VAR_GLOBAL CONSTANT  (* DbmDescriptions *)
  gc_DbmTranslation_de_Text0 : WSTRING(39) := "Pressure Block Oscillation Sensor State";
  gc_DbmTranslation_de_Text1 : WSTRING(39) := "Pressure Block Oscillation Sensor Value";
  gc_DbmTranslation_de_Text2 : WSTRING(43) := "Pressure Block Oscillation Sensor Raw value";
  gc_DbmTranslation_de_Text3 : WSTRING(27) := "Pressure Brake Sensor State";
  gc_DbmTranslation_de_Text4 : WSTRING(27) := "Pressure Brake Sensor Value";
  gc_DbmTranslation_de_Text5 : WSTRING(31) := "Pressure Brake Sensor Raw value";
  gc_DbmTranslation_de_Text6 : WSTRING(37) := "Temperature Transmission Sensor State";
  gc_DbmTranslation_de_Text7 : WSTRING(37) := "Temperature Transmission Sensor Value";
  gc_DbmTranslation_de_Text8 : WSTRING(41) := "Temperature Transmission Sensor Raw value";
  gc_DbmTranslation_de_Text9 : WSTRING(25) := "Fault Pvg Left Trak State";
  gc_DbmTranslation_de_Text10 : WSTRING(29) := "Fault Pvg Left Trak Raw Value";
  gc_DbmTranslation_de_Text11 : WSTRING(26) := "Fault Pvg Right Trak State";
  gc_DbmTranslation_de_Text12 : WSTRING(30) := "Fault Pvg Right Trak Raw value";
  gc_DbmTranslation_de_Text13 : WSTRING(25) := "Down Axle oscillant State";
  gc_DbmTranslation_de_Text14 : WSTRING(39) := "Down Axle oscillant  Raw value pin 0 Nc";
  gc_DbmTranslation_de_Text15 : WSTRING(39) := "Down Axle oscillant  Raw value pin 1 No";
  gc_DbmTranslation_de_Text16 : WSTRING(20) := "Down Axle fixe state";
  gc_DbmTranslation_de_Text17 : WSTRING(24) := "Down Axle fixe Raw value";
  gc_DbmTranslation_de_Text18 : WSTRING(33) := "Down Axle fixe Raw value pin 1 No";
  gc_DbmTranslation_de_Text19 : WSTRING(23) := "Up Axle oscillant state";
  gc_DbmTranslation_de_Text20 : WSTRING(23) := "Up Axle oscillant value";
  gc_DbmTranslation_de_Text21 : WSTRING(18) := "Up Axle fixe state";
  gc_DbmTranslation_de_Text22 : WSTRING(22) := "Up Axle fixe raw value";
  gc_DbmTranslation_de_Text23 : WSTRING(29) := "Frame rotation sensor 1 state";
  gc_DbmTranslation_de_Text24 : WSTRING(33) := "Frame rotation sensor 1 raw value";
  gc_DbmTranslation_de_Text25 : WSTRING(39) := "Frame rotation sensor 1 raw value Pin 1";
  gc_DbmTranslation_de_Text26 : WSTRING(22) := "Rail hook sensor state";
  gc_DbmTranslation_de_Text27 : WSTRING(26) := "Rail hook sensor raw value";
  gc_DbmTranslation_de_Text28 : WSTRING(27) := "Inductive Rail sensor state";
  gc_DbmTranslation_de_Text29 : WSTRING(31) := "Inductive Rail sensor raw value";
  gc_DbmTranslation_de_Text30 : WSTRING(21) := "Centered turret state";
  gc_DbmTranslation_de_Text31 : WSTRING(25) := "Centered turret raw value";
  gc_DbmTranslation_de_Text32 : WSTRING(25) := "Work Key track Side state";
  gc_DbmTranslation_de_Text33 : WSTRING(29) := "Work Key track Side raw value";
  gc_DbmTranslation_de_Text34 : WSTRING(29) := "Frame rotation sensor 2 state";
  gc_DbmTranslation_de_Text35 : WSTRING(39) := "Frame rotation sensor 2 raw value Pin 0";
  gc_DbmTranslation_de_Text36 : WSTRING(39) := "Frame rotation sensor 2 raw value Pin 1";
  gc_DbmTranslation_de_Text37 : WSTRING(24) := "Work Key Bilateral state";
  gc_DbmTranslation_de_Text38 : WSTRING(28) := "Work Key Bilateral raw value";
  gc_DbmTranslation_de_Text39 : WSTRING(22) := "Work Key Centred state";
  gc_DbmTranslation_de_Text40 : WSTRING(26) := "Work Key Centred raw value";
  gc_DbmTranslation_de_Text41 : WSTRING(32) := "Abutment turret track side state";
  gc_DbmTranslation_de_Text42 : WSTRING(36) := "Abutment turret track side raw value";
  gc_DbmTranslation_de_Text43 : WSTRING(34) := "Abutment Turret Centred Side state";
  gc_DbmTranslation_de_Text44 : WSTRING(38) := "Abutment Turret Centred Side raw value";
  gc_DbmTranslation_de_Text45 : WSTRING(43) := "Oscillant Axle Speed Sensor Direction state";
  gc_DbmTranslation_de_Text46 : WSTRING(47) := "Oscillant Axle Speed Sensor Direction Raw value";
  gc_DbmTranslation_de_Text47 : WSTRING(38) := "Fixe Axle Speed Sensor Direction state";
  gc_DbmTranslation_de_Text48 : WSTRING(42) := "Fixe Axle Speed Sensor Direction Raw value";
  gc_DbmTranslation_de_Text49 : WSTRING(19) := "Trailer gache state";
  gc_DbmTranslation_de_Text50 : WSTRING(23) := "Trailer gache raw value";
  gc_DbmTranslation_de_Text51 : WSTRING(34) := "Measuring mast sensor folded state";
  gc_DbmTranslation_de_Text52 : WSTRING(38) := "Measuring mast sensor folded raw value";
  gc_DbmTranslation_de_Text53 : WSTRING(24) := "Oscillant Axle frequency";
  gc_DbmTranslation_de_Text54 : WSTRING(19) := "Fixe Axle frequency";
  gc_DbmTranslation_de_Text55 : WSTRING(25) := "Aru Radio 1 Contact state";
  gc_DbmTranslation_de_Text56 : WSTRING(29) := "Aru Radio 1 Contact raw value";
  gc_DbmTranslation_de_Text57 : WSTRING(25) := "Aru Radio 2 Contact state";
  gc_DbmTranslation_de_Text58 : WSTRING(29) := "Aru Radio 2 Contact raw value";
  gc_DbmTranslation_de_Text59 : WSTRING(19) := "Aru 1 Contact state";
  gc_DbmTranslation_de_Text60 : WSTRING(23) := "Aru 1 Contact raw value";
  gc_DbmTranslation_de_Text61 : WSTRING(19) := "Aru 2 Contact state";
  gc_DbmTranslation_de_Text62 : WSTRING(23) := "Aru 2 contact raw value";
  gc_DbmTranslation_de_Text63 : WSTRING(19) := "Starter motor state";
  gc_DbmTranslation_de_Text64 : WSTRING(23) := "Starter motor raw value";
  gc_DbmTranslation_de_Text65 : WSTRING(33) := "Autorisation High Speed Key State";
  gc_DbmTranslation_de_Text66 : WSTRING(37) := "Autorisation High Speed Key Raw Value";
  gc_DbmTranslation_de_Text67 : WSTRING(35) := "Electric pump Pressure Sensor State";
  gc_DbmTranslation_de_Text68 : WSTRING(35) := "Electric pump Pressure Sensor Value";
  gc_DbmTranslation_de_Text69 : WSTRING(39) := "Electric pump Pressure Sensor Raw value";
  gc_DbmTranslation_de_Text70 : WSTRING(29) := "Mast sensor position UP State";
  gc_DbmTranslation_de_Text71 : WSTRING(33) := "Mast sensor position UP Raw Value";
  gc_DbmTranslation_de_Text72 : WSTRING(46) := "Hydraulic valve uin down position sensor state";
  gc_DbmTranslation_de_Text73 : WSTRING(50) := "Hydraulic valve uin down position sensor raw value";
  gc_DbmTranslation_de_Text74 : WSTRING(33) := "Ev Deflector Transmission command";
  gc_DbmTranslation_de_Text75 : WSTRING(38) := "Ev Deflector Transmission actual value";
  gc_DbmTranslation_de_Text76 : WSTRING(28) := "Ev Up Measuring Mast command";
  gc_DbmTranslation_de_Text77 : WSTRING(33) := "Ev Up Measuring Mast actual value";
  gc_DbmTranslation_de_Text78 : WSTRING(30) := "Ev Down Measuring Mast command";
  gc_DbmTranslation_de_Text79 : WSTRING(35) := "Ev Down Measuring Mast actual value";
  gc_DbmTranslation_de_Text80 : WSTRING(30) := "Ev Service Brake Track command";
  gc_DbmTranslation_de_Text81 : WSTRING(35) := "Ev Service Brake Track actual value";
  gc_DbmTranslation_de_Text82 : WSTRING(26) := "Ev Power Reduction command";
  gc_DbmTranslation_de_Text83 : WSTRING(31) := "Ev Power Reduction actual value";
  gc_DbmTranslation_de_Text84 : WSTRING(27) := "Ev Frame Rotation 1 command";
  gc_DbmTranslation_de_Text85 : WSTRING(32) := "Ev Frame Rotation 1 actual value";
  gc_DbmTranslation_de_Text86 : WSTRING(27) := "Ev Frame Rotation 2 command";
  gc_DbmTranslation_de_Text87 : WSTRING(32) := "Ev Frame Rotation 2 actual value";
  gc_DbmTranslation_de_Text88 : WSTRING(29) := "Supply Radio Receiver command";
  gc_DbmTranslation_de_Text89 : WSTRING(34) := "Supply Radio Receiver actual value";
  gc_DbmTranslation_de_Text90 : WSTRING(34) := "Buzzer Lynx Moving Machine command";
  gc_DbmTranslation_de_Text91 : WSTRING(39) := "Buzzer Lynx Moving Machine actual value";
  gc_DbmTranslation_de_Text92 : WSTRING(28) := "White Lights Trailer command";
  gc_DbmTranslation_de_Text93 : WSTRING(33) := "White Lights Trailer actual value";
  gc_DbmTranslation_de_Text94 : WSTRING(26) := "Red Lights Trailer command";
  gc_DbmTranslation_de_Text95 : WSTRING(31) := "Red Lights Trailer actual value";
  gc_DbmTranslation_de_Text96 : WSTRING(23) := "White Light AVG command";
  gc_DbmTranslation_de_Text97 : WSTRING(28) := "White Light AVG actual value";
  gc_DbmTranslation_de_Text98 : WSTRING(23) := "White Light AVD command";
  gc_DbmTranslation_de_Text99 : WSTRING(28) := "White Light AVD actual value";
  gc_DbmTranslation_de_Text100 : WSTRING(21) := "Red Light AVG command";
  gc_DbmTranslation_de_Text101 : WSTRING(26) := "Red Light AVG actual value";
  gc_DbmTranslation_de_Text102 : WSTRING(21) := "Red Light AVD command";
  gc_DbmTranslation_de_Text103 : WSTRING(26) := "Red Light AVD actual value";
  gc_DbmTranslation_de_Text104 : WSTRING(23) := "White Light ARG command";
  gc_DbmTranslation_de_Text105 : WSTRING(28) := "White Light ARG actual value";
  gc_DbmTranslation_de_Text106 : WSTRING(23) := "White Light ARD command";
  gc_DbmTranslation_de_Text107 : WSTRING(28) := "White Light ARD actual value";
  gc_DbmTranslation_de_Text108 : WSTRING(21) := "Red Light ARG command";
  gc_DbmTranslation_de_Text109 : WSTRING(26) := "Red Light ARG actual value";
  gc_DbmTranslation_de_Text110 : WSTRING(21) := "Red Light ARD command";
  gc_DbmTranslation_de_Text111 : WSTRING(26) := "Red Light ARD actual value";
  gc_DbmTranslation_de_Text112 : WSTRING(29) := "Suplly Pvg Left Track command";
  gc_DbmTranslation_de_Text113 : WSTRING(34) := "Suplly Pvg Left Track actual value";
  gc_DbmTranslation_de_Text114 : WSTRING(30) := "Suplly Pvg Right Track command";
  gc_DbmTranslation_de_Text115 : WSTRING(35) := "Suplly Pvg Right Track actual value";
  gc_DbmTranslation_de_Text116 : WSTRING(33) := "Ev UnBlock Oscillation Axle state";
  gc_DbmTranslation_de_Text117 : WSTRING(40) := "Ev UnBlock Oscillation Axle command bool";
  gc_DbmTranslation_de_Text118 : WSTRING(26) := "Ev Up Axle Oscillant state";
  gc_DbmTranslation_de_Text119 : WSTRING(33) := "Ev Up Axle Oscillant Command Bool";
  gc_DbmTranslation_de_Text120 : WSTRING(29) := "Ev Down Axle Oscillant  state";
  gc_DbmTranslation_de_Text121 : WSTRING(35) := "Ev Down Axle Oscillant Command Bool";
  gc_DbmTranslation_de_Text122 : WSTRING(20) := "Ev Up AxleFixe state";
  gc_DbmTranslation_de_Text123 : WSTRING(28) := "Ev Up Axle Fixe Command Bool";
  gc_DbmTranslation_de_Text124 : WSTRING(22) := "Ev Down AxleFixe state";
  gc_DbmTranslation_de_Text125 : WSTRING(30) := "Ev Down Axle Fixe Command Bool";
  gc_DbmTranslation_de_Text126 : WSTRING(35) := "Ev Park Brake Axle Oscillant  state";
  gc_DbmTranslation_de_Text127 : WSTRING(42) := "Ev Park Brake Axle Oscillant  command bool";
  gc_DbmTranslation_de_Text128 : WSTRING(29) := "Ev Park Brake Axle Fixe state";
  gc_DbmTranslation_de_Text129 : WSTRING(37) := "Ev Park Brake Axle Fixe  command bool";
  gc_DbmTranslation_de_Text130 : WSTRING(37) := "Ev Service Brake Axle Oscillant state";
  gc_DbmTranslation_de_Text131 : WSTRING(36) := "Ev Service Brake Axle 1 command Bool";
  gc_DbmTranslation_de_Text132 : WSTRING(32) := "Ev Service Brake Axle Fixe state";
  gc_DbmTranslation_de_Text133 : WSTRING(36) := "Ev Service Brake Axle 2 command Bool";
  gc_DbmTranslation_de_Text134 : WSTRING(19) := "Klaxon Neotec state";
  gc_DbmTranslation_de_Text135 : WSTRING(26) := "Klaxon Neotec command bool";
  gc_DbmTranslation_de_Text136 : WSTRING(18) := "Forward pump state";
  gc_DbmTranslation_de_Text137 : WSTRING(21) := "Forward pump  command";
  gc_DbmTranslation_de_Text138 : WSTRING(27) := "Forward pump actual current";
  gc_DbmTranslation_de_Text139 : WSTRING(19) := "Backward pump state";
  gc_DbmTranslation_de_Text140 : WSTRING(22) := "Backward pump  command";
  gc_DbmTranslation_de_Text141 : WSTRING(28) := "Backward pump actual current";
  gc_DbmTranslation_de_Text142 : WSTRING(22) := "Pvg left track command";
  gc_DbmTranslation_de_Text143 : WSTRING(29) := "Pvg left track actual voltage";
  gc_DbmTranslation_de_Text144 : WSTRING(23) := "Pvg right track command";
  gc_DbmTranslation_de_Text145 : WSTRING(30) := "Pvg right track actual voltage";
  gc_DbmTranslation_de_Text146 : WSTRING(26) := "Supply Ana Sensors Command";
  gc_DbmTranslation_de_Text147 : WSTRING(24) := "Supply Ana Sensors Value";
  gc_DbmTranslation_de_Text148 : WSTRING(30) := "Pvg Left Track Lowside Command";
  gc_DbmTranslation_de_Text149 : WSTRING(28) := "Pvg Left Track Lowside Value";
  gc_DbmTranslation_de_Text150 : WSTRING(31) := "Pvg Right Track Lowside Command";
  gc_DbmTranslation_de_Text151 : WSTRING(29) := "Pvg Right Track Lowside Value";
  gc_DbmTranslation_de_Text152 : WSTRING(39) := "Return low side Ev Forward Pump command";
  gc_DbmTranslation_de_Text153 : WSTRING(37) := "Return low side Ev Forward Pump state";
  gc_DbmTranslation_de_Text154 : WSTRING(40) := "Return low side Ev Backward Pump command";
  gc_DbmTranslation_de_Text155 : WSTRING(38) := "Return low side Ev Backward Pump state";
  gc_DbmTranslation_de_Text156 : WSTRING(19) := "Neon Lights command";
  gc_DbmTranslation_de_Text157 : WSTRING(17) := "Neon Lights value";
  gc_DbmTranslation_de_Text158 : WSTRING(33) := "Ev 2 Deflector Transmission value";
  gc_DbmTranslation_de_Text159 : WSTRING(21) := "Cooling relay command";
  gc_DbmTranslation_de_Text160 : WSTRING(19) := "Cooling relay state";
  gc_DbmTranslation_de_Text161 : WSTRING(54) := "Sorties d’activation de l’Ev du deuxième frein de parc";
  gc_DbmTranslation_de_Text162 : WSTRING(54) := "Sorties d’activation de l’Ev du deuxième frein de parc";
  gc_DbmTranslation_de_Text163 : WSTRING(33) := "Ev 2nd Park Brake Axle Fixe State";
  gc_DbmTranslation_de_Text164 : WSTRING(33) := "Ev 2nd Park Brake Axle Osci State";
  gc_DbmTranslation_de_Text165 : WSTRING(41) := "Pvg Translation for Rail Electric Command";
  gc_DbmTranslation_de_Text166 : WSTRING(41) := "Pvg Translation for Rail Electric Voltage";
  gc_DbmTranslation_de_Text167 : WSTRING(48) := "Suplly Pvg Translation for Rail Electric Command";
  gc_DbmTranslation_de_Text168 : WSTRING(46) := "Suplly Pvg Translation for Rail Electric State";
  gc_DbmTranslation_de_Text169 : WSTRING(42) := "Ev Deviator for Rail Electric Mode Command";
  gc_DbmTranslation_de_Text170 : WSTRING(40) := "Ev Deviator for Rail Electric Mode State";
  gc_DbmTranslation_de_Text171 : WSTRING(43) := "Relay Cut Off Variator for Electric Command";
  gc_DbmTranslation_de_Text172 : WSTRING(41) := "Relay Cut Off Variator for Electric State";
  gc_DbmTranslation_de_Text173 : WSTRING(28) := "Relay Enable Battery Command";
  gc_DbmTranslation_de_Text174 : WSTRING(26) := "Relay Enable Battery State";
  gc_DbmTranslation_de_Text175 : WSTRING(25) := "Byte increased each cycle";
  gc_DbmTranslation_de_Text176 : WSTRING(22) := "Watchdog current state";
  gc_DbmTranslation_de_Text177 : WSTRING(11) := "Ecu voltage";
  gc_DbmTranslation_de_Text178 : WSTRING(13) := "Off Rail Mode";
  gc_DbmTranslation_de_Text179 : WSTRING(9) := "Rail Mode";
  gc_DbmTranslation_de_Text180 : WSTRING(75) := "Output value Lut of Manipulator left radio control in range -10000 to 10000";
  gc_DbmTranslation_de_Text181 : WSTRING(35) := "Output value Lut of Left Track Pvg ";
  gc_DbmTranslation_de_Text182 : WSTRING(76) := "Output value Lut of Manipulator Right radio control in range -10000 to 10000";
  gc_DbmTranslation_de_Text183 : WSTRING(36) := "Output value Lut of Right Track Pvg ";
  gc_DbmTranslation_de_Text184 : WSTRING(52) := "Outût value Lut of Joystick advance Rail translation";
  gc_DbmTranslation_de_Text185 : WSTRING(40) := "Output Lut  of Forward Pump Transmission";
  gc_DbmTranslation_de_Text186 : WSTRING(41) := "Output Lut  of Backward Pump Transmission";
  gc_DbmTranslation_de_Text187 : WSTRING(71) := "Calculate consigne current of Forward Pump transmission on percent *100";
  gc_DbmTranslation_de_Text188 : WSTRING(24) := "LastJoystickAdvanceValue";
  gc_DbmTranslation_de_Text189 : WSTRING(37) := "Scaling Value of Joystick advancement";
  gc_DbmTranslation_de_Text190 : WSTRING(39) := "State of service brake rail translation";
  gc_DbmTranslation_de_Text191 : WSTRING(36) := "Enable Start timer for service brake";
  gc_DbmTranslation_de_Text192 : WSTRING(48) := "Speed motor command provide by track transaltion";
  gc_DbmTranslation_de_Text193 : WSTRING(28) := "Force silent mode motor test";
  gc_DbmTranslation_de_Text194 : WSTRING(19) := "Angular sensor test";
  gc_DbmTranslation_de_Text195 : WSTRING(17) := "Speed axle sensor";
  gc_DbmTranslation_de_Text196 : WSTRING(18) := "Average Time cycle";
  gc_DbmTranslation_de_Text197 : WSTRING(14) := "Max time cycle";
  gc_DbmTranslation_de_Text198 : WSTRING(40) := "First translation for release park brake";
  gc_DbmTranslation_de_Text199 : WSTRING(35) := "Autorize Up Axle Oscillant movement";
  gc_DbmTranslation_de_Text200 : WSTRING(37) := "Autorize Down Axle Oscillant movement";
  gc_DbmTranslation_de_Text201 : WSTRING(30) := "Autorize Up Axle fixe movement";
  gc_DbmTranslation_de_Text202 : WSTRING(32) := "Autorize Down Axle fixe movement";
  gc_DbmTranslation_de_Text203 : WSTRING(19) := "Engine On run phase";
  gc_DbmTranslation_de_Text204 : WSTRING(74) := "Transaltion rail or off rail is solicited , flag send to C1 to pilot motor";
  gc_DbmTranslation_de_Text205 : WSTRING(42) := "Direction of rail translation (Av Ar Stop)";
  gc_DbmTranslation_de_Text206 : WSTRING(39) := "Set condition to active Aru radio alarm";
  gc_DbmTranslation_de_Text207 : WSTRING(36) := "Joystick advance setpoint after ramp";
  gc_DbmTranslation_de_Text208 : WSTRING(46) := "Stabilized stop flag to active park brake rail";
  gc_DbmTranslation_de_Text209 : WSTRING(48) := "Emergency brake flag to active sequence of brake";
  gc_DbmTranslation_de_Text210 : WSTRING(51) := "Flag when the timer emergency service brake is done";
  gc_DbmTranslation_de_Text211 : WSTRING(66) := "Flag when the timer stopped machine unblock osciilant axle is done";
  gc_DbmTranslation_de_Text212 : WSTRING(86) := "Output value Lut of Manipulator left radio control in range -10000 to 10000 after ramp";
  gc_DbmTranslation_de_Text213 : WSTRING(87) := "Output value Lut of Manipulator right radio control in range -10000 to 10000 after ramp";
  gc_DbmTranslation_de_Text214 : WSTRING(52) := "Delta beetwen left and right Pvg crawler advancement";
  gc_DbmTranslation_de_Text215 : WSTRING(65) := "Consigne left pvg track calcul with delta beetween left and right";
  gc_DbmTranslation_de_Text216 : WSTRING(66) := "Consigne right pvg track calcul with delta beetween left and right";
  gc_DbmTranslation_de_Text217 : WSTRING(56) := "Flag to detect brake when gachette or pedal are released";
  gc_DbmTranslation_de_Text218 : WSTRING(50) := "Counter for debug when alarm aru radio is detected";
  gc_DbmTranslation_de_Text219 : WSTRING(28) := "Red light ARG basket command";
  gc_DbmTranslation_de_Text220 : WSTRING(30) := "White light ARG basket command";
  gc_DbmTranslation_de_Text221 : WSTRING(32) := "Portilon close and ladder folded";
  gc_DbmTranslation_de_Text222 : WSTRING(46) := "Test boolean  command to refresh objet evision";
  gc_DbmTranslation_de_Text223 : WSTRING(60) := "Position of joysstick advancment ( AV_JOY, NEU_JOY , AR_JOY)";
  gc_DbmTranslation_de_Text224 : WSTRING(81) := "Retain position of joystick advancement , reset when brake sequence is sollicited";
  gc_DbmTranslation_de_Text225 : WSTRING(37) := "Authorize forward crawler translation";
  gc_DbmTranslation_de_Text226 : WSTRING(38) := "Authorize backward crawler translation";
  gc_DbmTranslation_de_Text227 : WSTRING(22) := "Return value uart init";
  gc_DbmTranslation_de_Text228 : WSTRING(35) := "Authorize translation rail movement";
  gc_DbmTranslation_de_Text229 : WSTRING(25) := "Ev forward track consigne";
  gc_DbmTranslation_de_Text230 : WSTRING(24) := "Ev forward rail consigne";
  gc_DbmTranslation_de_Text231 : WSTRING(0) := "";
  gc_DbmTranslation_de_Text232 : WSTRING(21) := "Variable debug Neotec";
  gc_DbmTranslation_de_Text233 : WSTRING(21) := "Variable debug Neotec";
  gc_DbmTranslation_de_Text234 : WSTRING(21) := "Variable debug Neotec";
  gc_DbmTranslation_de_Text235 : WSTRING(21) := "Variable debug Neotec";
  gc_DbmTranslation_de_Text236 : WSTRING(21) := "Variable debug Neotec";
  gc_DbmTranslation_de_Text237 : WSTRING(21) := "Variable debug Neotec";
  gc_DbmTranslation_de_Text238 : WSTRING(21) := "Variable debug Neotec";
  gc_DbmTranslation_de_Text239 : WSTRING(21) := "Variable debug Neotec";
  gc_DbmTranslation_de_Text240 : WSTRING(21) := "Variable debug Neotec";
  gc_DbmTranslation_de_Text241 : WSTRING(21) := "Variable debug Neotec";
  gc_DbmTranslation_de_Text242 : WSTRING(21) := "Variable debug Neotec";
  gc_DbmTranslation_de_Text243 : WSTRING(21) := "Variable debug Neotec";
  gc_DbmTranslation_de_Text244 : WSTRING(21) := "Variable debug Neotec";
  gc_DbmTranslation_de_Text245 : WSTRING(21) := "Variable debug Neotec";
  gc_DbmTranslation_de_Text246 : WSTRING(21) := "Variable debug Neotec";
  gc_DbmTranslation_de_Text247 : WSTRING(21) := "Variable debug Neotec";
  gc_DbmTranslation_de_Text248 : WSTRING(21) := "Variable debug Neotec";
  gc_DbmTranslation_de_Text249 : WSTRING(21) := "Variable debug Neotec";
  gc_DbmTranslation_de_Text250 : WSTRING(21) := "Variable debug Neotec";
  gc_DbmTranslation_de_Text251 : WSTRING(21) := "Variable debug Neotec";
  gc_DbmTranslation_de_Text252 : WSTRING(21) := "Variable debug Neotec";
  gc_DbmTranslation_de_Text253 : WSTRING(21) := "Variable debug Neotec";
  gc_DbmTranslation_de_Text254 : WSTRING(21) := "Variable debug Neotec";
  gc_DbmTranslation_de_Text255 : WSTRING(21) := "Variable debug Neotec";
  gc_DbmTranslation_de_Text256 : WSTRING(21) := "Variable debug Neotec";
  gc_DbmTranslation_de_Text257 : WSTRING(21) := "Variable debug Neotec";
  gc_DbmTranslation_de_Text258 : WSTRING(21) := "Variable debug Neotec";
  gc_DbmTranslation_de_Text259 : WSTRING(21) := "Variable debug Neotec";
  gc_DbmTranslation_de_Text260 : WSTRING(21) := "Variable debug Neotec";
  gc_DbmTranslation_de_Text261 : WSTRING(21) := "Variable debug Neotec";
  gc_DbmTranslation_de_Text262 : WSTRING(21) := "Variable debug Neotec";
  gc_DbmTranslation_de_Text263 : WSTRING(21) := "Variable debug Neotec";
  gc_DbmTranslation_de_Text264 : WSTRING(21) := "Variable debug Neotec";
  gc_DbmTranslation_de_Text265 : WSTRING(21) := "Variable debug Neotec";
  gc_DbmTranslation_de_Text266 : WSTRING(21) := "Variable debug Neotec";
  gc_DbmTranslation_de_Text267 : WSTRING(21) := "Variable debug Neotec";
  gc_DbmTranslation_de_Text268 : WSTRING(21) := "Variable debug Neotec";
  gc_DbmTranslation_de_Text269 : WSTRING(21) := "Variable debug Neotec";
  gc_DbmTranslation_de_Text270 : WSTRING(21) := "Variable debug Neotec";
  gc_DbmTranslation_de_Text271 : WSTRING(21) := "Variable debug Neotec";
  gc_DbmTranslation_de_Text272 : WSTRING(28) := "Red light ARD basket command";
  gc_DbmTranslation_de_Text273 : WSTRING(30) := "White light ARD basket command";
  gc_DbmTranslation_de_Text274 : WSTRING(26) := "Active failure is detected";
  gc_DbmTranslation_de_Text275 : WSTRING(19) := "Reduction pump rail";
  gc_DbmTranslation_de_Text276 : WSTRING(20) := "Reduction pump track";
  gc_DbmTranslation_de_Text277 : WSTRING(25) := "Active white lights 15746";
  gc_DbmTranslation_de_Text278 : WSTRING(24) := "White light Av 15746 Cmd";
  gc_DbmTranslation_de_Text279 : WSTRING(24) := "White light Ar 15746 Cmd";
  gc_DbmTranslation_de_Text280 : WSTRING(38) := "Shunt all logic to test electricall IO";
  gc_DbmTranslation_de_Text281 : WSTRING(29) := "Send Event Datalogger Message";
  gc_DbmTranslation_de_Text282 : WSTRING(21) := "Depend de l’option MG";
  gc_DbmTranslation_de_Text283 : WSTRING(13) := "Slow Blinking";
  gc_DbmTranslation_de_Text284 : WSTRING(14) := "Total distance";
  gc_DbmTranslation_de_Text285 : WSTRING(19) := "Running Stable 48XS";
  gc_DbmTranslation_de_Text286 : WSTRING(39) := "Alarm Hydraulic Temperature Rail Active";
  gc_DbmTranslation_de_Text287 : WSTRING(42) := "Alarm Hydraulic Temperature Crawler Active";
  gc_DbmTranslation_de_Text288 : WSTRING(17) := "Diag Faulty Value";
  gc_DbmTranslation_de_Text289 : WSTRING(15) := "Diag Device Num";
  gc_DbmTranslation_de_Text290 : WSTRING(15) := "Diag Error Code";
  gc_DbmTranslation_de_Text291 : WSTRING(21) := "Engine running stable";
  gc_DbmTranslation_de_Text292 : WSTRING(42) := "Select config hollandaise to control light";
  gc_DbmTranslation_de_Text293 : WSTRING(37) := "Portillon is installed on the machine";
  gc_DbmTranslation_de_Text294 : WSTRING(34) := "Ladder is installed on the machine";
  gc_DbmTranslation_de_Text295 : WSTRING(41) := "Measuring mat is installed on the machine";
  gc_DbmTranslation_de_Text296 : WSTRING(107) := "-SpeedMaxRail Acces Site- Inclinaison Baslet most be in low sector for acces site speed on translation rail";
  gc_DbmTranslation_de_Text297 : WSTRING(90) := "-SpeedMaxRail Acces Site- Basket most be centered for acces site speed on translation rail";
  gc_DbmTranslation_de_Text298 : WSTRING(64) := "The digital display o the measuring mast is used on this vehicle";
  gc_DbmTranslation_de_Text299 : WSTRING(30) := "Autorisation work key present ";
  gc_DbmTranslation_de_Text300 : WSTRING(40) := "Option d’activation du mode double frein";
  gc_DbmTranslation_de_Text301 : WSTRING(50) := "Strukton configuration for new performance machine";
  gc_DbmTranslation_de_Text302 : WSTRING(46) := "Basket and turret limited by a mechanical stop";
  gc_DbmTranslation_de_Text303 : WSTRING(24) := "Presence of sensor plate";
  gc_DbmTranslation_de_Text304 : WSTRING(29) := "Number of brake cycle perform";
  gc_DbmTranslation_de_Text305 : WSTRING(10) := "Light mode";
  gc_DbmTranslation_de_Text306 : WSTRING(0) := "";
  gc_DbmTranslation_de_Text307 : WSTRING(0) := "";
  gc_DbmTranslation_de_Text308 : WSTRING(0) := "";
  gc_DbmTranslation_de_Text309 : WSTRING(0) := "";
  gc_DbmTranslation_de_Text310 : WSTRING(0) := "";
  gc_DbmTranslation_de_Text311 : WSTRING(0) := "";
  gc_DbmTranslation_de_Text312 : WSTRING(0) := "";
  gc_DbmTranslation_de_Text313 : WSTRING(0) := "";
  gc_DbmTranslation_de_Text314 : WSTRING(0) := "";
  gc_DbmTranslation_de_Text315 : WSTRING(0) := "";
  gc_DbmTranslation_de_Text316 : WSTRING(0) := "";
  gc_DbmTranslation_de_Text317 : WSTRING(0) := "";
  gc_DbmTranslation_de_Text318 : WSTRING(0) := "";
  gc_DbmTranslation_de_Text319 : WSTRING(0) := "";
  gc_DbmTranslation_de_Text320 : WSTRING(0) := "";
  gc_DbmTranslation_de_Text321 : WSTRING(54) := "Nombres de cycle de frein pour les freins additionnels";
  gc_DbmTranslation_de_Text322 : WSTRING(18) := "Total Distance Msb";
  gc_DbmTranslation_de_Text323 : WSTRING(18) := "Total Distance Lsb";
  gc_DbmTranslation_de_Text324 : WSTRING(77) := "Limit threshold of angle to stop movement , angular sensor from radio control";
  gc_DbmTranslation_de_Text325 : WSTRING(43) := "Treshold minimal speed to active park brake";
  gc_DbmTranslation_de_Text326 : WSTRING(46) := "Treshold minimal speed to active service brake";
  gc_DbmTranslation_de_Text327 : WSTRING(41) := "Additionnal Pourcent Forward Pump Command";
  gc_DbmTranslation_de_Text328 : WSTRING(67) := "Additionnal Pourcent Forward Pump Command when sient mode is active";
  gc_DbmTranslation_de_Text329 : WSTRING(21) := "Node Id radio command";
  gc_DbmTranslation_de_Text330 : WSTRING(34) := "Dead Zone joystick rotation turret";
  gc_DbmTranslation_de_Text331 : WSTRING(52) := "Timer before 2nd Service Axle brake rail translation";
  gc_DbmTranslation_de_Text332 : WSTRING(26) := "Time Service Brake Offrail";
  gc_DbmTranslation_de_Text333 : WSTRING(59) := "Ev Forward Pump - PWM output parameters- engine off current";
  gc_DbmTranslation_de_Text334 : WSTRING(56) := "Ev Forward Pump - PWM output parameters- minimal current";
  gc_DbmTranslation_de_Text335 : WSTRING(54) := "Ev Forward Pump - PWM output parameters- stop current ";
  gc_DbmTranslation_de_Text336 : WSTRING(60) := "Ev Backward Pump - PWM output parameters- engine off current";
  gc_DbmTranslation_de_Text337 : WSTRING(57) := "Ev Backward Pump - PWM output parameters- minimal current";
  gc_DbmTranslation_de_Text338 : WSTRING(55) := "Ev Backward Pump - PWM output parameters- stop current ";
  gc_DbmTranslation_de_Text339 : WSTRING(67) := "Position neutral of joystick advancement regarding batterie voltage";
  gc_DbmTranslation_de_Text340 : WSTRING(46) := "PID - Ev Forward Pump - Gp - proportional gain";
  gc_DbmTranslation_de_Text341 : WSTRING(54) := "PID - Ev Forward Pump - Ti - integration time constant";
  gc_DbmTranslation_de_Text342 : WSTRING(53) := "PID - Ev Forward Pump - Td - derivation time constant";
  gc_DbmTranslation_de_Text343 : WSTRING(46) := "PID - Ev Forward Pump - Gp - proportional gain";
  gc_DbmTranslation_de_Text344 : WSTRING(54) := "PID - Ev Forward Pump - Ti - integration time constant";
  gc_DbmTranslation_de_Text345 : WSTRING(53) := "PID - Ev Forward Pump - Td - derivation time constant";
  gc_DbmTranslation_de_Text346 : WSTRING(80) := "PressureBlockOscillationSensor - input current - output characteristic - Positif";
  gc_DbmTranslation_de_Text347 : WSTRING(80) := "PressureBlockOscillationSensor - input current - output characteristic - Neutral";
  gc_DbmTranslation_de_Text348 : WSTRING(80) := "PressureBlockOscillationSensor - input current - output characteristic - Negatif";
  gc_DbmTranslation_de_Text349 : WSTRING(69) := "PressureBrakeSensor - input current - output characteristic - Positif";
  gc_DbmTranslation_de_Text350 : WSTRING(69) := "PressureBrakeSensor - input current - output characteristic - Neutral";
  gc_DbmTranslation_de_Text351 : WSTRING(69) := "PressureBrakeSensor - input current - output characteristic - Negatif";
  gc_DbmTranslation_de_Text352 : WSTRING(79) := "TemperatureTransmissionSensor - input current - output characteristic - Positif";
  gc_DbmTranslation_de_Text353 : WSTRING(79) := "TemperatureTransmissionSensor - input current - output characteristic - Neutral";
  gc_DbmTranslation_de_Text354 : WSTRING(79) := "TemperatureTransmissionSensor - input current - output characteristic - Negatif";
  gc_DbmTranslation_de_Text355 : WSTRING(55) := "Consigne min Ev forward apply with joystick advancement";
  gc_DbmTranslation_de_Text356 : WSTRING(55) := "Consigne max Ev forward apply with joystick advancement";
  gc_DbmTranslation_de_Text357 : WSTRING(56) := "Consigne min Ev backward apply with joystick advancement";
  gc_DbmTranslation_de_Text358 : WSTRING(56) := "Consigne max Ev backward apply with joystick advancement";
  gc_DbmTranslation_de_Text359 : WSTRING(96) := "Time  ramp to Ev rail [0] Pos incr time, [1] Pos decr time,[2] Neg incr time , [3] Neg decr time";
  gc_DbmTranslation_de_Text360 : WSTRING(96) := "Time  ramp to Ev rail [0] Pos incr time, [1] Pos decr time,[2] Neg incr time , [3] Neg decr time";
  gc_DbmTranslation_de_Text361 : WSTRING(96) := "Time  ramp to Ev rail [0] Pos incr time, [1] Pos decr time,[2] Neg incr time , [3] Neg decr time";
  gc_DbmTranslation_de_Text362 : WSTRING(96) := "Time  ramp to Ev rail [0] Pos incr time, [1] Pos decr time,[2] Neg incr time , [3] Neg decr time";
  gc_DbmTranslation_de_Text363 : WSTRING(96) := "Time  ramp to Ev rail [0] Pos incr time, [1] Pos decr time,[2] Neg incr time , [3] Neg decr time";
  gc_DbmTranslation_de_Text364 : WSTRING(53) := "Consigne min Ev forward apply for crawler advancement";
  gc_DbmTranslation_de_Text365 : WSTRING(53) := "Consigne max Ev forward apply for crawler advancement";
  gc_DbmTranslation_de_Text366 : WSTRING(72) := "Ratio apply to ramp signal to control Ev forward for crawler advancement";
  gc_DbmTranslation_de_Text367 : WSTRING(72) := "Ratio apply to ramp signal to control Ev forward for crawler advancement";
  gc_DbmTranslation_de_Text368 : WSTRING(72) := "Ratio apply to ramp signal to control Ev forward for crawler advancement";
  gc_DbmTranslation_de_Text369 : WSTRING(69) := "Park Brake rail - Treshold of regime motor to active park brake rail ";
  gc_DbmTranslation_de_Text370 : WSTRING(95) := "Consigne min Pvg Left Track apply when mapinulator get out neutral position to forward position";
  gc_DbmTranslation_de_Text371 : WSTRING(30) := "Consigne max Pvg Left Track Av";
  gc_DbmTranslation_de_Text372 : WSTRING(96) := "Consigne min Pvg Left Track apply when mapinulator get out neutral position to backward position";
  gc_DbmTranslation_de_Text373 : WSTRING(30) := "Consigne max Pvg Left Track Ar";
  gc_DbmTranslation_de_Text374 : WSTRING(96) := "Consigne min Pvg Right Track apply when mapinulator get out neutral position to forward position";
  gc_DbmTranslation_de_Text375 : WSTRING(31) := "Consigne max Pvg Right Track Av";
  gc_DbmTranslation_de_Text376 : WSTRING(97) := "Consigne min Pvg Right Track apply when mapinulator get out neutral position to backward position";
  gc_DbmTranslation_de_Text377 : WSTRING(31) := "Consigne max Pvg Right Track Ar";
  gc_DbmTranslation_de_Text378 : WSTRING(105) := "Time  ramp apply to left track [0] Pos incr time, [1] Pos decr time,[2] Neg incr time , [3] Neg decr time";
  gc_DbmTranslation_de_Text379 : WSTRING(105) := "Time  ramp apply to left track [0] Pos incr time, [1] Pos decr time,[2] Neg incr time , [3] Neg decr time";
  gc_DbmTranslation_de_Text380 : WSTRING(105) := "Time  ramp apply to left track [0] Pos incr time, [1] Pos decr time,[2] Neg incr time , [3] Neg decr time";
  gc_DbmTranslation_de_Text381 : WSTRING(105) := "Time  ramp apply to left track [0] Pos incr time, [1] Pos decr time,[2] Neg incr time , [3] Neg decr time";
  gc_DbmTranslation_de_Text382 : WSTRING(105) := "Time  ramp apply to left track [0] Pos incr time, [1] Pos decr time,[2] Neg incr time , [3] Neg decr time";
  gc_DbmTranslation_de_Text383 : WSTRING(106) := "Time  ramp apply to right track [0] Pos incr time, [1] Pos decr time,[2] Neg incr time , [3] Neg decr time";
  gc_DbmTranslation_de_Text384 : WSTRING(106) := "Time  ramp apply to right track [0] Pos incr time, [1] Pos decr time,[2] Neg incr time , [3] Neg decr time";
  gc_DbmTranslation_de_Text385 : WSTRING(106) := "Time  ramp apply to right track [0] Pos incr time, [1] Pos decr time,[2] Neg incr time , [3] Neg decr time";
  gc_DbmTranslation_de_Text386 : WSTRING(106) := "Time  ramp apply to right track [0] Pos incr time, [1] Pos decr time,[2] Neg incr time , [3] Neg decr time";
  gc_DbmTranslation_de_Text387 : WSTRING(106) := "Time  ramp apply to right track [0] Pos incr time, [1] Pos decr time,[2] Neg incr time , [3] Neg decr time";
  gc_DbmTranslation_de_Text388 : WSTRING(38) := "Time to detect stabilized stop machine";
  gc_DbmTranslation_de_Text389 : WSTRING(67) := "Treshold low spped to start timer to detect stabilized stop machine";
  gc_DbmTranslation_de_Text390 : WSTRING(66) := "Time before release service brake when emergency brake is detected";
  gc_DbmTranslation_de_Text391 : WSTRING(57) := "Time stopped machine to controle unblock oscillation axle";
  gc_DbmTranslation_de_Text392 : WSTRING(87) := "Low treshold speed of oscillation and fixe axle to start timer unblock oscillation axle";
  gc_DbmTranslation_de_Text393 : WSTRING(55) := "Gap max beetween left and right Pvg crawler advancement";
  gc_DbmTranslation_de_Text394 : WSTRING(84) := "Gap max beetween left and right Pvg crawler advancement when manipulator is inverted";
  gc_DbmTranslation_de_Text395 : WSTRING(36) := "Treshold Ana to bool input from 48xs";
  gc_DbmTranslation_de_Text396 : WSTRING(65) := "In min joystick advancement pourcentent by 10 of batterie voltage";
  gc_DbmTranslation_de_Text397 : WSTRING(65) := "In max joystick advancement pourcentent by 10 of batterie voltage";
  gc_DbmTranslation_de_Text398 : WSTRING(35) := "Speed mini treshol to re authorise ";
  gc_DbmTranslation_de_Text399 : WSTRING(44) := "Number element for average slope trans angle";
  gc_DbmTranslation_de_Text400 : WSTRING(43) := "Number element for average slope long angle";
  gc_DbmTranslation_de_Text401 : WSTRING(35) := "Dead zone joystick rail advancement";
  gc_DbmTranslation_de_Text402 : WSTRING(57) := "Number element for average slope trans angle 2nd channels";
  gc_DbmTranslation_de_Text403 : WSTRING(56) := "Number element for average slope long angle 2nd channels";
  gc_DbmTranslation_de_Text404 : WSTRING(18) := "Param debug Neotec";
  gc_DbmTranslation_de_Text405 : WSTRING(18) := "Param debug Neotec";
  gc_DbmTranslation_de_Text406 : WSTRING(18) := "Param debug Neotec";
  gc_DbmTranslation_de_Text407 : WSTRING(18) := "Param debug Neotec";
  gc_DbmTranslation_de_Text408 : WSTRING(18) := "Param debug Neotec";
  gc_DbmTranslation_de_Text409 : WSTRING(18) := "Param debug Neotec";
  gc_DbmTranslation_de_Text410 : WSTRING(18) := "Param debug Neotec";
  gc_DbmTranslation_de_Text411 : WSTRING(18) := "Param debug Neotec";
  gc_DbmTranslation_de_Text412 : WSTRING(18) := "Param debug Neotec";
  gc_DbmTranslation_de_Text413 : WSTRING(18) := "Param debug Neotec";
  gc_DbmTranslation_de_Text414 : WSTRING(18) := "Param debug Neotec";
  gc_DbmTranslation_de_Text415 : WSTRING(18) := "Param debug Neotec";
  gc_DbmTranslation_de_Text416 : WSTRING(18) := "Param debug Neotec";
  gc_DbmTranslation_de_Text417 : WSTRING(18) := "Param debug Neotec";
  gc_DbmTranslation_de_Text418 : WSTRING(18) := "Param debug Neotec";
  gc_DbmTranslation_de_Text419 : WSTRING(18) := "Param debug Neotec";
  gc_DbmTranslation_de_Text420 : WSTRING(18) := "Param debug Neotec";
  gc_DbmTranslation_de_Text421 : WSTRING(57) := "Treshold hydraulique temperature to control cooling relay";
  gc_DbmTranslation_de_Text422 : WSTRING(22) := "Time to control cooler";
  gc_DbmTranslation_de_Text423 : WSTRING(37) := "Time fault pressure reduction crawler";
  gc_DbmTranslation_de_Text424 : WSTRING(35) := "Rail joystick ratio two speed fault";
  gc_DbmTranslation_de_Text425 : WSTRING(25) := "Timeout sdo resquest time";
  gc_DbmTranslation_de_Text426 : WSTRING(29) := "Period Blinck off White Light";
  gc_DbmTranslation_de_Text427 : WSTRING(48) := "filtrage et le lissage de la valeur du joystick.";
  gc_DbmTranslation_de_Text428 : WSTRING(92) := "temporisation de l’AU afin d’attendre la fin des rampes avec un freinage d’urgence (Mode MG)";
  gc_DbmTranslation_de_Text429 : WSTRING(59) := "seuil d’angle tourelle pour la petite vitesse, côté positif";
  gc_DbmTranslation_de_Text430 : WSTRING(59) := "seuil d’angle tourelle pour la petite vitesse, côté négatif";
  gc_DbmTranslation_de_Text431 : WSTRING(25) := "Number of file parameters";
  gc_DbmTranslation_de_Text432 : WSTRING(13) := "Version Major";
  gc_DbmTranslation_de_Text433 : WSTRING(14) := "Version Minior";
  gc_DbmTranslation_de_Text434 : WSTRING(13) := "Version Patch";
  gc_DbmTranslation_de_Text435 : WSTRING(14) := "Version Custom";
  gc_DbmTranslation_de_Text436 : WSTRING(76) := "ElectricPumpPressureSensor - input current - output characteristic - Positif";
  gc_DbmTranslation_de_Text437 : WSTRING(76) := "ElectricPumpPressureSensor - input current - output characteristic - Neutral";
  gc_DbmTranslation_de_Text438 : WSTRING(76) := "ElectricPumpPressureSensor - input current - output characteristic - Negatif";
  gc_DbmTranslation_de_Text439 : WSTRING(44) := "Max point Lut Manipulator Left radio control";
  gc_DbmTranslation_de_Text440 : WSTRING(52) := "Lut array X value for Manipulator Left radio control";
  gc_DbmTranslation_de_Text441 : WSTRING(52) := "Lut array X value for Manipulator Left radio control";
  gc_DbmTranslation_de_Text442 : WSTRING(52) := "Lut array X value for Manipulator Left radio control";
  gc_DbmTranslation_de_Text443 : WSTRING(52) := "Lut array Y value for Manipulator Left radio control";
  gc_DbmTranslation_de_Text444 : WSTRING(52) := "Lut array Y value for Manipulator Left radio control";
  gc_DbmTranslation_de_Text445 : WSTRING(52) := "Lut array Y value for Manipulator Left radio control";
  gc_DbmTranslation_de_Text446 : WSTRING(45) := "Max point Lut Manipulator Right radio control";
  gc_DbmTranslation_de_Text447 : WSTRING(53) := "Lut array X value for Manipulator Right radio control";
  gc_DbmTranslation_de_Text448 : WSTRING(53) := "Lut array X value for Manipulator Right radio control";
  gc_DbmTranslation_de_Text449 : WSTRING(53) := "Lut array X value for Manipulator Right radio control";
  gc_DbmTranslation_de_Text450 : WSTRING(53) := "Lut array Y value for Manipulator Right radio control";
  gc_DbmTranslation_de_Text451 : WSTRING(53) := "Lut array Y value for Manipulator Right radio control";
  gc_DbmTranslation_de_Text452 : WSTRING(53) := "Lut array Y value for Manipulator Right radio control";
  gc_DbmTranslation_de_Text453 : WSTRING(40) := "Max point Lut for Left track pvg command";
  gc_DbmTranslation_de_Text454 : WSTRING(25) := "Left track Pvg Ramp ratio";
  gc_DbmTranslation_de_Text455 : WSTRING(25) := "Left track Pvg Ramp ratio";
  gc_DbmTranslation_de_Text456 : WSTRING(25) := "Left track Pvg Ramp ratio";
  gc_DbmTranslation_de_Text457 : WSTRING(50) := "Range value of left track Pvg apply to ramp signal";
  gc_DbmTranslation_de_Text458 : WSTRING(50) := "Range value of left track Pvg apply to ramp signal";
  gc_DbmTranslation_de_Text459 : WSTRING(50) := "Range value of left track Pvg apply to ramp signal";
  gc_DbmTranslation_de_Text460 : WSTRING(50) := "Range value of left track Pvg apply to ramp signal";
  gc_DbmTranslation_de_Text461 : WSTRING(26) := "Right track Pvg Ramp ratio";
  gc_DbmTranslation_de_Text462 : WSTRING(26) := "Right track Pvg Ramp ratio";
  gc_DbmTranslation_de_Text463 : WSTRING(26) := "Right track Pvg Ramp ratio";
  gc_DbmTranslation_de_Text464 : WSTRING(51) := "Range value of right track Pvg apply to ramp signal";
  gc_DbmTranslation_de_Text465 : WSTRING(51) := "Range value of right track Pvg apply to ramp signal";
  gc_DbmTranslation_de_Text466 : WSTRING(51) := "Range value of right track Pvg apply to ramp signal";
  gc_DbmTranslation_de_Text467 : WSTRING(51) := "Range value of right track Pvg apply to ramp signal";
  gc_DbmTranslation_de_Text468 : WSTRING(56) := "Max point Lut Forward pump transmission rail translation";
  gc_DbmTranslation_de_Text469 : WSTRING(64) := "Lut array X value for Forward pump transmission rail translation";
  gc_DbmTranslation_de_Text470 : WSTRING(64) := "Lut array X value for Forward pump transmission rail translation";
  gc_DbmTranslation_de_Text471 : WSTRING(64) := "Lut array X value for Forward pump transmission rail translation";
  gc_DbmTranslation_de_Text472 : WSTRING(64) := "Lut array Y value for Forward pump transmission rail translation";
  gc_DbmTranslation_de_Text473 : WSTRING(64) := "Lut array Y value for Forward pump transmission rail translation";
  gc_DbmTranslation_de_Text474 : WSTRING(64) := "Lut array Y value for Forward pump transmission rail translation";
  gc_DbmTranslation_de_Text475 : WSTRING(57) := "Max point Lut Backward pump transmission rail translation";
  gc_DbmTranslation_de_Text476 : WSTRING(64) := "Lut array X value for Backwardpump transmission rail translation";
  gc_DbmTranslation_de_Text477 : WSTRING(64) := "Lut array X value for Backwardpump transmission rail translation";
  gc_DbmTranslation_de_Text478 : WSTRING(64) := "Lut array X value for Backwardpump transmission rail translation";
  gc_DbmTranslation_de_Text479 : WSTRING(64) := "Lut array Y value for Backwardpump transmission rail translation";
  gc_DbmTranslation_de_Text480 : WSTRING(64) := "Lut array Y value for Backwardpump transmission rail translation";
  gc_DbmTranslation_de_Text481 : WSTRING(64) := "Lut array Y value for Backwardpump transmission rail translation";
  gc_DbmTranslation_de_Text482 : WSTRING(36) := "Forward pump transmission Ramp ratio";
  gc_DbmTranslation_de_Text483 : WSTRING(36) := "Forward pump transmission Ramp ratio";
  gc_DbmTranslation_de_Text484 : WSTRING(36) := "Forward pump transmission Ramp ratio";
  gc_DbmTranslation_de_Text485 : WSTRING(51) := "Range value of Forward pump transmission Ramp ratio";
  gc_DbmTranslation_de_Text486 : WSTRING(51) := "Range value of Forward pump transmission Ramp ratio";
  gc_DbmTranslation_de_Text487 : WSTRING(51) := "Range value of Forward pump transmission Ramp ratio";
  gc_DbmTranslation_de_Text488 : WSTRING(51) := "Range value of Forward pump transmission Ramp ratio";
  gc_DbmTranslation_de_Text489 : WSTRING(37) := "Backward pump transmission Ramp ratio";
  gc_DbmTranslation_de_Text490 : WSTRING(37) := "Backward pump transmission Ramp ratio";
  gc_DbmTranslation_de_Text491 : WSTRING(37) := "Backward pump transmission Ramp ratio";
  gc_DbmTranslation_de_Text492 : WSTRING(52) := "Range value of Backward pump transmission Ramp ratio";
  gc_DbmTranslation_de_Text493 : WSTRING(52) := "Range value of Backward pump transmission Ramp ratio";
  gc_DbmTranslation_de_Text494 : WSTRING(52) := "Range value of Backward pump transmission Ramp ratio";
  gc_DbmTranslation_de_Text495 : WSTRING(52) := "Range value of Backward pump transmission Ramp ratio";
  gc_DbmTranslation_de_Text496 : WSTRING(38) := "Offset apply to calcul angle of turret";
  gc_DbmTranslation_de_Text497 : WSTRING(55) := "Slope Long offset to calibrate value of longetude angle";
  gc_DbmTranslation_de_Text498 : WSTRING(58) := "Slope Trans offset to calibrate value of transversal angle";
  gc_DbmTranslation_de_Text499 : WSTRING(68) := "Slope Long offset to calibrate value of longetude angle 2nd channels";
  gc_DbmTranslation_de_Text500 : WSTRING(71) := "Slope Trans offset to calibrate value of transversal angle 2nd channels";
  gc_DbmTranslation_de_Text501 : WSTRING(53) := "Offset apply to calcul angle of turret second channel";
  gc_DbmTranslation_de_Text502 : WSTRING(21) := "Encodeur Turret Msb 1";
  gc_DbmTranslation_de_Text503 : WSTRING(21) := "Encodeur Turret Msb 2";
  gc_DbmTranslation_de_Text504 : WSTRING(21) := "Encodeur Turret Lsb 1";
  gc_DbmTranslation_de_Text505 : WSTRING(21) := "Encodeur Turret Lsb 2";
  gc_DbmTranslation_de_Text506 : WSTRING(29) := "Up  Inclinaison basket button";
  gc_DbmTranslation_de_Text507 : WSTRING(40) := "Up  Inclinaison basket  button raw value";
  gc_DbmTranslation_de_Text508 : WSTRING(31) := "Down  Inclinaison basket button";
  gc_DbmTranslation_de_Text509 : WSTRING(41) := "Down  Inclinaison basket button raw value";
  gc_DbmTranslation_de_Text510 : WSTRING(18) := "Up pendular button";
  gc_DbmTranslation_de_Text511 : WSTRING(28) := "Up pendular button raw value";
  gc_DbmTranslation_de_Text512 : WSTRING(20) := "Down pendular button";
  gc_DbmTranslation_de_Text513 : WSTRING(30) := "Down pendular button raw value";
  gc_DbmTranslation_de_Text514 : WSTRING(40) := "Counter Clockwise rotation basket button";
  gc_DbmTranslation_de_Text515 : WSTRING(50) := "Counter Clockwise rotation basket button raw value";
  gc_DbmTranslation_de_Text516 : WSTRING(32) := "Clockwise rotation basket button";
  gc_DbmTranslation_de_Text517 : WSTRING(42) := "Clockwise rotation basket button raw value";
  gc_DbmTranslation_de_Text518 : WSTRING(10) := "Overload 1";
  gc_DbmTranslation_de_Text519 : WSTRING(20) := "Overload 1 raw value";
  gc_DbmTranslation_de_Text520 : WSTRING(10) := "Overload 2";
  gc_DbmTranslation_de_Text521 : WSTRING(20) := "Overload 2 raw value";
  gc_DbmTranslation_de_Text522 : WSTRING(34) := "Nacelle basket right side sensor 1";
  gc_DbmTranslation_de_Text523 : WSTRING(40) := "Nacelle basket right side sensor 1 value";
  gc_DbmTranslation_de_Text524 : WSTRING(35) := "Nacelle basket right side sensor 2 ";
  gc_DbmTranslation_de_Text525 : WSTRING(40) := "Nacelle basket right side sensor 2 value";
  gc_DbmTranslation_de_Text526 : WSTRING(33) := "Nacelle basket left side sensor 1";
  gc_DbmTranslation_de_Text527 : WSTRING(39) := "Nacelle basket left side sensor 1 value";
  gc_DbmTranslation_de_Text528 : WSTRING(33) := "Nacelle basket left side sensor 2";
  gc_DbmTranslation_de_Text529 : WSTRING(39) := "Nacelle basket left side sensor 2 value";
  gc_DbmTranslation_de_Text530 : WSTRING(26) := "Low sector pendular sensor";
  gc_DbmTranslation_de_Text531 : WSTRING(32) := "Low sector pendular sensor value";
  gc_DbmTranslation_de_Text532 : WSTRING(24) := "High Sector Plate Sensor";
  gc_DbmTranslation_de_Text533 : WSTRING(30) := "High Sector Plate Sensor value";
  gc_DbmTranslation_de_Text534 : WSTRING(20) := "Folded ladder sensor";
  gc_DbmTranslation_de_Text535 : WSTRING(26) := "Folded ladder sensor value";
  gc_DbmTranslation_de_Text536 : WSTRING(23) := "Safety man system value";
  gc_DbmTranslation_de_Text537 : WSTRING(29) := "Delta arm axis joystick value";
  gc_DbmTranslation_de_Text538 : WSTRING(29) := "Arrow arm axis joystick value";
  gc_DbmTranslation_de_Text539 : WSTRING(33) := "Telescope arm axis joystick value";
  gc_DbmTranslation_de_Text540 : WSTRING(35) := "Rotation turret axis joystick value";
  gc_DbmTranslation_de_Text541 : WSTRING(27) := "Advance axis joystick value";
  gc_DbmTranslation_de_Text542 : WSTRING(28) := "Rearmement Safety Man System";
  gc_DbmTranslation_de_Text543 : WSTRING(34) := "Rearmement Safety Man System value";
  gc_DbmTranslation_de_Text544 : WSTRING(28) := "Abutement Nacelle Track Side";
  gc_DbmTranslation_de_Text545 : WSTRING(34) := "Abutement Nacelle Track Side value";
  gc_DbmTranslation_de_Text546 : WSTRING(31) := "Abutement Nacelle Centered Side";
  gc_DbmTranslation_de_Text547 : WSTRING(37) := "Abutement Nacelle Centered Side value";
  gc_DbmTranslation_de_Text548 : WSTRING(24) := "Delta arm Joystick value";
  gc_DbmTranslation_de_Text549 : WSTRING(38) := "Arrow Joystick / centered turret value";
  gc_DbmTranslation_de_Text550 : WSTRING(31) := "Centered advance joystick value";
  gc_DbmTranslation_de_Text551 : WSTRING(20) := "Dead man pedal value";
  gc_DbmTranslation_de_Text552 : WSTRING(35) := "Pressence in nacelle sensor 1 value";
  gc_DbmTranslation_de_Text553 : WSTRING(35) := "Pressence in nacelle sensor 2 value";
  gc_DbmTranslation_de_Text554 : WSTRING(14) := "Gachette value";
  gc_DbmTranslation_de_Text555 : WSTRING(12) := "Klaxon value";
  gc_DbmTranslation_de_Text556 : WSTRING(17) := "Stop Motor button";
  gc_DbmTranslation_de_Text557 : WSTRING(28) := "Authorization work key value";
  gc_DbmTranslation_de_Text558 : WSTRING(27) := "Etallonnage Joystick Button";
  gc_DbmTranslation_de_Text559 : WSTRING(22) := "Close Portillon Sensor";
  gc_DbmTranslation_de_Text560 : WSTRING(31) := "Heartbeat for slave module 48xs";
  gc_DbmTranslation_de_Text561 : WSTRING(37) := "Batterie voltage of module slave 48xs";
  gc_DbmTranslation_de_Text562 : WSTRING(20) := "White Lights command";
  gc_DbmTranslation_de_Text563 : WSTRING(25) := "White Lights actual value";
  gc_DbmTranslation_de_Text564 : WSTRING(18) := "Red Lights command";
  gc_DbmTranslation_de_Text565 : WSTRING(23) := "Red Lights actual value";
  gc_DbmTranslation_de_Text566 : WSTRING(18) := "Work Light command";
  gc_DbmTranslation_de_Text567 : WSTRING(18) := "Work Light command";
  gc_DbmTranslation_de_Text568 : WSTRING(14) := "Buzzer command";
  gc_DbmTranslation_de_Text569 : WSTRING(19) := "Buzzer actual value";
  gc_DbmTranslation_de_Text570 : WSTRING(41) := "Error status of Motor Default Light ouput";
  gc_DbmTranslation_de_Text571 : WSTRING(36) := "Error status of Overload Light ouput";
  gc_DbmTranslation_de_Text572 : WSTRING(28) := "Error status of Buzzer ouput";
  gc_DbmTranslation_de_Text573 : WSTRING(35) := "Error status of Gas Oil Light ouput";
  gc_DbmTranslation_de_Text574 : WSTRING(42) := "Error status of devers default light ouput";
  gc_DbmTranslation_de_Text575 : WSTRING(35) := "Error status of Red Light ARD ouput";
  gc_DbmTranslation_de_Text576 : WSTRING(43) := "Error status of White Light ARD light ouput";
  gc_DbmTranslation_de_Text577 : WSTRING(35) := "Error status of Warming Light ouput";
  gc_DbmTranslation_de_Text578 : WSTRING(35) := "Error status of Red Light ARG ouput";
  gc_DbmTranslation_de_Text579 : WSTRING(43) := "Error status of White Light ARG light ouput";
  gc_DbmTranslation_de_Text580 : WSTRING(22) := "State of radio control";
  gc_DbmTranslation_de_Text581 : WSTRING(16) := "Left manipulator";
  gc_DbmTranslation_de_Text582 : WSTRING(17) := "Right manipulator";
  gc_DbmTranslation_de_Text583 : WSTRING(23) := "LeftManipulatorPosition";
  gc_DbmTranslation_de_Text584 : WSTRING(24) := "RightManipulatorPosition";
  gc_DbmTranslation_de_Text585 : WSTRING(12) := "UpAxleArFixe";
  gc_DbmTranslation_de_Text586 : WSTRING(14) := "DownAxleArFixe";
  gc_DbmTranslation_de_Text587 : WSTRING(17) := "UpAxleAvOscillant";
  gc_DbmTranslation_de_Text588 : WSTRING(19) := "DownAxleAvOscillant";
  gc_DbmTranslation_de_Text589 : WSTRING(32) := "Rotation frame Coutner clockwise";
  gc_DbmTranslation_de_Text590 : WSTRING(24) := "Rotation frame clockwise";
  gc_DbmTranslation_de_Text591 : WSTRING(24) := "Selector rotation turret";
  gc_DbmTranslation_de_Text592 : WSTRING(17) := "Selector pendular";
  gc_DbmTranslation_de_Text593 : WSTRING(21) := "Radio command connect";
  gc_DbmTranslation_de_Text594 : WSTRING(40) := "Up pendular or rotation clockwise turret";
  gc_DbmTranslation_de_Text595 : WSTRING(50) := "down pendular or rotation counter clockwise turret";
  gc_DbmTranslation_de_Text596 : WSTRING(19) := "Start radio command";
  gc_DbmTranslation_de_Text597 : WSTRING(18) := "Stop radio command";
  gc_DbmTranslation_de_Text598 : WSTRING(21) := "Forcing advance track";
  gc_DbmTranslation_de_Text599 : WSTRING(14) := "Klaxon command";
  gc_DbmTranslation_de_Text600 : WSTRING(27) := "Encodeur turret 1 angle raw";
  gc_DbmTranslation_de_Text601 : WSTRING(51) := "Encodeur turret 1 angle with calibration parameters";
  gc_DbmTranslation_de_Text602 : WSTRING(27) := "Encodeur turret 2 angle raw";
  gc_DbmTranslation_de_Text603 : WSTRING(51) := "Encodeur turret 2 angle with calibration parameters";
  gc_DbmTranslation_de_Text604 : WSTRING(26) := "Devers1 X axis angle value";
  gc_DbmTranslation_de_Text605 : WSTRING(26) := "Devers1 Y axis angle value";
  gc_DbmTranslation_de_Text606 : WSTRING(46) := "Slope Long Angle value with calibration offset";
  gc_DbmTranslation_de_Text607 : WSTRING(47) := "Slope Trans Angle value with calibration offset";
  gc_DbmTranslation_de_Text608 : WSTRING(30) := "State heart beat devers sensor";
  gc_DbmTranslation_de_Text609 : WSTRING(41) := "State heart beat encodeur turret sensor 1";
  gc_DbmTranslation_de_Text610 : WSTRING(20) := "Selected slope angle";
  gc_DbmTranslation_de_Text611 : WSTRING(31) := "Encodeur mast measure raw value";
  gc_DbmTranslation_de_Text612 : WSTRING(62) := "Encodeur mast measure with calibration parameters in centilmer";
  gc_DbmTranslation_de_Text613 : WSTRING(26) := "Devers2 X axis angle value";
  gc_DbmTranslation_de_Text614 : WSTRING(26) := "Devers2 Y axis angle value";
  gc_DbmTranslation_de_Text615 : WSTRING(28) := "Slope Alarm 1 receive by CAN";
  gc_DbmTranslation_de_Text616 : WSTRING(28) := "Slope Alarm 2 receive by CAN";
  gc_DbmTranslation_de_Text617 : WSTRING(48) := "Slope Long Angle value with calibration offset 2";
  gc_DbmTranslation_de_Text618 : WSTRING(49) := "Slope Trans Angle value with calibration offset 2";
  gc_DbmTranslation_de_Text619 : WSTRING(51) := "Error code form emergency message encodeur turret 1";
  gc_DbmTranslation_de_Text620 : WSTRING(55) := "Error register form emergency message encodeur turret 1";
  gc_DbmTranslation_de_Text621 : WSTRING(51) := "Error code form emergency message encodeur turret 2";
  gc_DbmTranslation_de_Text622 : WSTRING(55) := "Error register form emergency message encodeur turret 2";
  gc_DbmTranslation_de_Text623 : WSTRING(46) := "Error code form emergency message mast measure";
  gc_DbmTranslation_de_Text624 : WSTRING(50) := "Error register form emergency message mast measure";
  gc_DbmTranslation_de_Text625 : WSTRING(41) := "State heart beat encodeur turret sensor 2";
  gc_DbmTranslation_de_Text626 : WSTRING(46) := "Timeout Sdo Request Detected Encodeur Turret 1";
  gc_DbmTranslation_de_Text627 : WSTRING(46) := "Timeout Sdo Request Detected Encodeur Turret 2";
  gc_DbmTranslation_de_Text628 : WSTRING(31) := "Encodeur turret calibrate value";
  gc_DbmTranslation_de_Text629 : WSTRING(33) := "Encodeur turret calibrate value 2";
  gc_DbmTranslation_de_Text630 : WSTRING(29) := "User Log in Status (1=log in)";
  gc_DbmTranslation_de_Text631 : WSTRING(21) := "Movement Allow Status";
  gc_DbmTranslation_de_Text632 : WSTRING(20) := "Break Parking Status";
  gc_DbmTranslation_de_Text633 : WSTRING(21) := "Break Faillure Status";
  gc_DbmTranslation_de_Text634 : WSTRING(23) := "Turret Sector in Center";
  gc_DbmTranslation_de_Text635 : WSTRING(23) := "Turret Sector in Center";
  gc_DbmTranslation_de_Text636 : WSTRING(37) := "Vehicule in Train Mode (Speed in MPH)";
  gc_DbmTranslation_de_Text637 : WSTRING(55) := "Incoherence between Lateral Stop and Key selector (A47)";
  gc_DbmTranslation_de_Text638 : WSTRING(44) := "0=Work Mode activate 1=Site Acces Mode  (A4)";
  gc_DbmTranslation_de_Text639 : WSTRING(35) := "Safety Electric Pump Activate (A44)";
  gc_DbmTranslation_de_Text640 : WSTRING(38) := "Downhill between 150mm and 200mm (A13)";
  gc_DbmTranslation_de_Text641 : WSTRING(22) := "Train Mode Allow (A10)";
  gc_DbmTranslation_de_Text642 : WSTRING(34) := "Brake test need to be launch (A22)";
  gc_DbmTranslation_de_Text643 : WSTRING(26) := "Brake Pressure Fault (A14)";
  gc_DbmTranslation_de_Text644 : WSTRING(29) := "Activate Measuring Mast (A21)";
  gc_DbmTranslation_de_Text645 : WSTRING(35) := "Auto Movement Direction Light (A23)";
  gc_DbmTranslation_de_Text646 : WSTRING(38) := "Back Railway Axle in Low Position (A7)";
  gc_DbmTranslation_de_Text647 : WSTRING(39) := "Front Railway Axle in Low Position (A7)";
  gc_DbmTranslation_de_Text648 : WSTRING(37) := "Back Railway Axle Service Brake (A25)";
  gc_DbmTranslation_de_Text649 : WSTRING(38) := "Front Railway Axle Service Brake (A25)";
  gc_DbmTranslation_de_Text650 : WSTRING(34) := "Back Railway Axle Park Brake (A26)";
  gc_DbmTranslation_de_Text651 : WSTRING(36) := "Front Railway Axle Park Brake (A26) ";
  gc_DbmTranslation_de_Text652 : WSTRING(43) := "Status of Front Left Train Brake Test (A27)";
  gc_DbmTranslation_de_Text653 : WSTRING(44) := "Status of Front Right Train Brake Test (A27)";
  gc_DbmTranslation_de_Text654 : WSTRING(42) := "Status of Back Left Train Brake Test (A27)";
  gc_DbmTranslation_de_Text655 : WSTRING(42) := "Status of Back Left Train Brake Test (A27)";
  gc_DbmTranslation_de_Text656 : WSTRING(23) := "Status of the ARU alarm";
  gc_DbmTranslation_de_Text657 : WSTRING(23) := "Engine use time in hour";
  gc_DbmTranslation_de_Text658 : WSTRING(10) := "Engine RPM";
  gc_DbmTranslation_de_Text659 : WSTRING(28) := "Vehicule Speed in Km/h * 100";
  gc_DbmTranslation_de_Text660 : WSTRING(72) := "Lateralization Stop 1=bi lateralization 2=ALO Work 3=Multiple track (A3)";
  gc_DbmTranslation_de_Text661 : WSTRING(64) := "Key Selector 1=bi lateralization 2=ALO Work 3=Multiple track(A6)";
  gc_DbmTranslation_de_Text662 : WSTRING(38) := "Front Speed Railway Axle in Km/h (A24)";
  gc_DbmTranslation_de_Text663 : WSTRING(31) := "Back Speed Railway Axle in Km/h";
  gc_DbmTranslation_de_Text664 : WSTRING(59) := "Button for the calibration of the turret encoder is pressed";
  gc_DbmTranslation_de_Text665 : WSTRING(47) := "Status of off track variable on test brake page";
  gc_DbmTranslation_de_Text666 : WSTRING(51) := "Status of off track variable on run in process page";
  gc_DbmTranslation_de_Text667 : WSTRING(41) := "Request status of osci service test brake";
  gc_DbmTranslation_de_Text668 : WSTRING(42) := "Request status of fixed service test brake";
  gc_DbmTranslation_de_Text669 : WSTRING(41) := "Request status of both service test brake";
  gc_DbmTranslation_de_Text670 : WSTRING(38) := "Request status of osci park test brake";
  gc_DbmTranslation_de_Text671 : WSTRING(39) := "Request status of fixed park test brake";
  gc_DbmTranslation_de_Text672 : WSTRING(38) := "Request status of both park test brake";
  gc_DbmTranslation_de_Text673 : WSTRING(43) := "Request status of osci service run in brake";
  gc_DbmTranslation_de_Text674 : WSTRING(49) := "Request status of fixed service run in test brake";
  gc_DbmTranslation_de_Text675 : WSTRING(48) := "Request status of both service run in test brake";
  gc_DbmTranslation_de_Text676 : WSTRING(35) := "Test brake page is active on screen";
  gc_DbmTranslation_de_Text677 : WSTRING(39) := "break in brake page is active on screen";
  gc_DbmTranslation_de_Text678 : WSTRING(13) := "Serial Number";
  gc_DbmTranslation_de_Text679 : WSTRING(18) := "BP Basket Validate";
  gc_DbmTranslation_de_Text680 : WSTRING(19) := "Key Filter Overload";
  gc_DbmTranslation_de_Text681 : WSTRING(13) := "Key Next Mode";
  gc_DbmTranslation_de_Text682 : WSTRING(13) := "Key Prev Mode";
  gc_DbmTranslation_de_Text683 : WSTRING(17) := "Key Signal Danger";
  gc_DbmTranslation_de_Text684 : WSTRING(18) := "Key Flash Light ON";
  gc_DbmTranslation_de_Text685 : WSTRING(18) := "Key Calib Mast Min";
  gc_DbmTranslation_de_Text686 : WSTRING(18) := "Key Calib Mast Max";
  gc_DbmTranslation_de_Text687 : WSTRING(17) := "KeyCalibMastValid";
  gc_DbmTranslation_de_Text688 : WSTRING(24) := "Key Generator Activation";
  gc_DbmTranslation_de_Text689 : WSTRING(40) := "raz distance travaled mast mesure button";
  gc_DbmTranslation_de_Text690 : WSTRING(22) := "Key white lights 15746";
  gc_DbmTranslation_de_Text691 : WSTRING(26) := "Osci 2nd Park Brake Select";
  gc_DbmTranslation_de_Text692 : WSTRING(26) := "Fixe 2nd Park Brake Select";
  gc_DbmTranslation_de_Text693 : WSTRING(18) := "RAZ controller Key";
  gc_DbmTranslation_de_Text694 : WSTRING(29) := "Turret post selector input C1";
  gc_DbmTranslation_de_Text695 : WSTRING(28) := "Radio Post Selector input C1";
  gc_DbmTranslation_de_Text696 : WSTRING(30) := "Nacelle Post Selector input C1";
  gc_DbmTranslation_de_Text697 : WSTRING(25) := "Up axle oscillant command";
  gc_DbmTranslation_de_Text698 : WSTRING(27) := "Down axle oscillant command";
  gc_DbmTranslation_de_Text699 : WSTRING(20) := "Up axle Fixe command";
  gc_DbmTranslation_de_Text700 : WSTRING(21) := "Down axle Fixecommand";
  gc_DbmTranslation_de_Text701 : WSTRING(27) := "Regime motor alternator rpm";
  gc_DbmTranslation_de_Text702 : WSTRING(26) := "Entry telescope fdc sensor";
  gc_DbmTranslation_de_Text703 : WSTRING(23) := "DElta arm folded sensor";
  gc_DbmTranslation_de_Text704 : WSTRING(23) := "Booom Arm folded sensor";
  gc_DbmTranslation_de_Text705 : WSTRING(23) := "Delta ram in lower zone";
  gc_DbmTranslation_de_Text706 : WSTRING(30) := "Arrow arm angular sensor value";
  gc_DbmTranslation_de_Text707 : WSTRING(33) := "Turret is in the rear center zone";
  gc_DbmTranslation_de_Text708 : WSTRING(34) := "Turret is in the front center zone";
  gc_DbmTranslation_de_Text709 : WSTRING(47) := "Folded delta arm zone detect with analog sensor";
  gc_DbmTranslation_de_Text710 : WSTRING(47) := "Folded arrow arm zone detect with analog sensor";
  gc_DbmTranslation_de_Text711 : WSTRING(21) := "No movement is during";
  gc_DbmTranslation_de_Text712 : WSTRING(30) := "Delta arm angular sensor value";
  gc_DbmTranslation_de_Text713 : WSTRING(31) := "Folded position of mast measure";
  gc_DbmTranslation_de_Text714 : WSTRING(22) := "Transmission1 Pressure";
  gc_DbmTranslation_de_Text715 : WSTRING(22) := "Transmission2 Pressure";
  gc_DbmTranslation_de_Text716 : WSTRING(17) := "Active Help state";
  gc_DbmTranslation_de_Text717 : WSTRING(25) := "Basket un center position";
  gc_DbmTranslation_de_Text718 : WSTRING(31) := "Stop all movements Nacelle post";
  gc_DbmTranslation_de_Text719 : WSTRING(39) := "Encodeur Mast measure value in centimer";
  gc_DbmTranslation_de_Text720 : WSTRING(41) := "Flag when mast measure function is active";
  gc_DbmTranslation_de_Text721 : WSTRING(34) := "Out of range transmission pressure";
  gc_DbmTranslation_de_Text722 : WSTRING(21) := "Commande du gyrophare";
  gc_DbmTranslation_de_Text723 : WSTRING(13) := "Moteur allumé";
  gc_DbmTranslation_de_Text724 : WSTRING(27) := "Alarme du capteur téléscope";
  gc_DbmTranslation_de_Text725 : WSTRING(30) := "Alarme sur le capteur tourelle";
  gc_DbmTranslation_de_Text726 : WSTRING(26) := "Option White Light EN15746";
  gc_DbmTranslation_de_Text727 : WSTRING(15) := "Safe man system";
  gc_DbmTranslation_de_Text728 : WSTRING(18) := "Slope Mode from C1";
  gc_DbmTranslation_de_Text729 : WSTRING(25) := "Cold Oil Tank Temperature";
  gc_DbmTranslation_de_Text730 : WSTRING(24) := "Electric Motor Forbidden";
  gc_DbmTranslation_de_Text731 : WSTRING(19) := "Rpm Electric Motor ";
  gc_DbmTranslation_de_Text732 : WSTRING(21) := "Oil Tank Temperature ";
  gc_DbmTranslation_de_Text733 : WSTRING(21) := "SOC stop regeneration";
  gc_DbmTranslation_de_Text734 : WSTRING(12) := "Generator ON";
  gc_DbmTranslation_de_Text735 : WSTRING(36) := "Active EV deviator movements command";
  gc_DbmTranslation_de_Text736 : WSTRING(23) := "Test electrical from C1";
  gc_DbmTranslation_de_Text737 : WSTRING(23) := "Automatic Mode Activate";
  gc_DbmTranslation_de_Text738 : WSTRING(21) := "Silence Mode Activate";
  gc_DbmTranslation_de_Text739 : WSTRING(30) := "Forcing Regeneration low level";
  gc_DbmTranslation_de_Text740 : WSTRING(31) := "Forcing Regeneration High level";
  gc_DbmTranslation_de_Text741 : WSTRING(17) := "EV Bypass command";
  gc_DbmTranslation_de_Text742 : WSTRING(21) := "Motor speed CMD J1939";
  gc_DbmTranslation_de_Text743 : WSTRING(50) := "Command to perform the calibration of turret angle";
  gc_DbmTranslation_de_Text744 : WSTRING(64) := "Command to perform the calibration of turret angle intermediaire";
  gc_DbmTranslation_de_Text745 : WSTRING(53) := "Command to perform the calibration of longetude angle";
  gc_DbmTranslation_de_Text746 : WSTRING(55) := "Command to perform the calibration of transversal angle";
  gc_DbmTranslation_de_Text747 : WSTRING(49) := "Command to saved calibration list value on EEPROM";
  gc_DbmTranslation_de_Text748 : WSTRING(52) := "Acces chantier speed aplly to consigne max EvForward";
  gc_DbmTranslation_de_Text749 : WSTRING(42) := "High speed aplly to consigne max EvForward";
  gc_DbmTranslation_de_Text750 : WSTRING(41) := "Low speed aplly to consigne max EvForward";
  gc_DbmTranslation_de_Text751 : WSTRING(67) := "Low speed apply to consigne max EvForward when test brake is needed";
  gc_DbmTranslation_de_Text752 : WSTRING(55) := "Treshold slope vehicule angle for high speed (absolute)";
  gc_DbmTranslation_de_Text753 : WSTRING(72) := "Hysteresis applied on the slope vehicule angle for high speed (relative)";
  gc_DbmTranslation_de_Text754 : WSTRING(54) := "Treshold slope vehicule angle for low speed (absolute)";
  gc_DbmTranslation_de_Text755 : WSTRING(71) := "Hysteresis applied on the slope vehicule angle for low speed (relative)";
  gc_DbmTranslation_de_Text756 : WSTRING(93) := "Treshold angle of turret for low speed in (relative to TurretRear PosFront and NegFront zone)";
  gc_DbmTranslation_de_Text757 : WSTRING(64) := "Hysteresis applied on the Treshold angle of turret for low speed";
  gc_DbmTranslation_de_Text758 : WSTRING(34) := "Rear center position of the turret";
  gc_DbmTranslation_de_Text759 : WSTRING(61) := "Front center position of the turret in the positive direction";
  gc_DbmTranslation_de_Text760 : WSTRING(61) := "Front center position of the turret in the negative direction";
  gc_DbmTranslation_de_Text761 : WSTRING(65) := "Limit speed on mode acces site speed wich trigger emergency brake";
  gc_DbmTranslation_de_Text762 : WSTRING(58) := "Limit speed on mode highSpeed wich trigger emergency brake";
  gc_DbmTranslation_de_Text763 : WSTRING(63) := "Limit speed on mode lowSpeed speed wich trigger emergency brake";
  gc_DbmTranslation_de_Text764 : WSTRING(69) := "Limit speed on mode Low Speed Brake Test wich trigger emergency brake";
  gc_DbmTranslation_de_Text765 : WSTRING(52) := "Acces chantier speed aplly to consigne max Backward ";
  gc_DbmTranslation_de_Text766 : WSTRING(42) := "High speed aplly to consigne max Backward ";
  gc_DbmTranslation_de_Text767 : WSTRING(41) := "Low speed aplly to consigne max Backward ";
  gc_DbmTranslation_de_Text768 : WSTRING(68) := "Low speed apply to consigne max EvBackward when test brake is needed";
  gc_DbmTranslation_de_Text769 : WSTRING(49) := "Test brake speed apply to consinge max Ev forward";
  gc_DbmTranslation_de_Text770 : WSTRING(50) := "Test brake speed apply to consinge max Ev backward";
  gc_DbmTranslation_de_Text771 : WSTRING(53) := "Break in brake speed apply to consinge max Ev forward";
  gc_DbmTranslation_de_Text772 : WSTRING(54) := "Break in brake speed apply to consinge max Ev backward";
  gc_DbmTranslation_de_Text773 : WSTRING(25) := "Arm speed rail hysteresis";
  gc_DbmTranslation_de_Text774 : WSTRING(36) := "Arm low sector basket fault treshold";
  gc_DbmTranslation_de_Text775 : WSTRING(26) := "Arm low zone for low speed";
  gc_DbmTranslation_de_Text776 : WSTRING(38) := "Turret rear negatif low speed treshold";
  gc_DbmTranslation_de_Text777 : WSTRING(38) := "Turret rear positif low speed treshold";
  gc_DbmTranslation_de_Text778 : WSTRING(33) := "Slope thres of 2 deg for STRUKTON";
  gc_DbmTranslation_de_Text779 : WSTRING(33) := "Slope thres of 4 deg for STRUKTON";
  gc_DbmTranslation_de_Text780 : WSTRING(33) := "Slope thres of 6 deg for STRUKTON";
  gc_DbmTranslation_de_Text781 : WSTRING(38) := "Slope Hyst for measure of slope angle ";
  gc_DbmTranslation_de_Text782 : WSTRING(51) := "Turret Hyst for sector of turret versus slope angle";
  gc_DbmTranslation_de_Text783 : WSTRING(41) := "Turret Sector for Slope angle below 2 Deg";
  gc_DbmTranslation_de_Text784 : WSTRING(62) := "Turret Sector for Slope angle below 2 Deg with rotation basket";
  gc_DbmTranslation_de_Text785 : WSTRING(41) := "Turret Sector for Slope angle below 4 Deg";
  gc_DbmTranslation_de_Text786 : WSTRING(62) := "Turret Sector for Slope angle below 4 Deg with rotation basket";
  gc_DbmTranslation_de_Text787 : WSTRING(41) := "Turret Sector for Slope angle below 6 Deg";
  gc_DbmTranslation_de_Text788 : WSTRING(62) := "Turret Sector for Slope angle below 6 Deg with rotation basket";
  gc_DbmTranslation_de_Text789 : WSTRING(60) := "Parameters to Prevention for Limit Speed in Acces Site Speed";
  gc_DbmTranslation_de_Text790 : WSTRING(54) := "Parameters to Prevention for Limit Speed in High Speed";
  gc_DbmTranslation_de_Text791 : WSTRING(53) := "Parameters to Prevention for Limit Speed in Low Speed";
  gc_DbmTranslation_de_Text792 : WSTRING(58) := "Parameters to Prevention for Speed in Low Speed Brake Test";
  gc_DbmTranslation_de_Text793 : WSTRING(76) := "Slope is over at high speed treshold (a hysteris is applied on the treshold)";
  gc_DbmTranslation_de_Text794 : WSTRING(76) := "Slope is lower at low speed treshold (a hysteris is applied on the treshold)";
  gc_DbmTranslation_de_Text795 : WSTRING(35) := "Turret angle in low speed rear zone";
  gc_DbmTranslation_de_Text796 : WSTRING(44) := "Turret angle in low speed postiif front zone";
  gc_DbmTranslation_de_Text797 : WSTRING(44) := "Turret angle in low speed negatif front zone";
  gc_DbmTranslation_de_Text798 : WSTRING(30) := "Turret angle in low speed zone";
  gc_DbmTranslation_de_Text799 : WSTRING(80) := "Enable simulation mode (use the simulation variables instead of the real inputs)";
  gc_DbmTranslation_de_Text800 : WSTRING(0) := "";
  gc_DbmTranslation_de_Text801 : WSTRING(0) := "";
  gc_DbmTranslation_de_Text802 : WSTRING(0) := "";
  gc_DbmTranslation_de_Text803 : WSTRING(0) := "";
  gc_DbmTranslation_de_Text804 : WSTRING(0) := "";
  gc_DbmTranslation_de_Text805 : WSTRING(0) := "";
  gc_DbmTranslation_de_Text806 : WSTRING(0) := "";
  gc_DbmTranslation_de_Text807 : WSTRING(0) := "";
  gc_DbmTranslation_de_Text808 : WSTRING(0) := "";
  gc_DbmTranslation_de_Text809 : WSTRING(0) := "";
  gc_DbmTranslation_de_Text810 : WSTRING(0) := "";
  gc_DbmTranslation_de_Text811 : WSTRING(0) := "";
  gc_DbmTranslation_de_Text812 : WSTRING(0) := "";
  gc_DbmTranslation_de_Text813 : WSTRING(0) := "";
  gc_DbmTranslation_de_Text814 : WSTRING(0) := "";
  gc_DbmTranslation_de_Text815 : WSTRING(0) := "";
  gc_DbmTranslation_de_Text816 : WSTRING(0) := "";
  gc_DbmTranslation_de_Text817 : WSTRING(0) := "";
  gc_DbmTranslation_de_Text818 : WSTRING(0) := "";
  gc_DbmTranslation_de_Text819 : WSTRING(49) := "Flag to detect exceeded of limit speed acces site";
  gc_DbmTranslation_de_Text820 : WSTRING(43) := "Flag to detect exceeded of limit speed high";
  gc_DbmTranslation_de_Text821 : WSTRING(48) := "Flag to detect exceeded of limit speed low speed";
  gc_DbmTranslation_de_Text822 : WSTRING(55) := "Flag to detect exceeded of limit speed speed brake test";
  gc_DbmTranslation_de_Text823 : WSTRING(32) := "Flag when one Litmit is exceeded";
  gc_DbmTranslation_de_Text824 : WSTRING(21) := "Kinematic train allow";
  gc_DbmTranslation_de_Text825 : WSTRING(31) := "Case of Slope angle below 2 deg";
  gc_DbmTranslation_de_Text826 : WSTRING(31) := "Case of Slope angle below 4 deg";
  gc_DbmTranslation_de_Text827 : WSTRING(31) := "Case of Slope angle below 6 deg";
  gc_DbmTranslation_de_Text828 : WSTRING(37) := "Case of Slope angle higher than 6 deg";
  gc_DbmTranslation_de_Text829 : WSTRING(36) := "Turret in Low Speed zone below 2 deg";
  gc_DbmTranslation_de_Text830 : WSTRING(36) := "Turret in Low Speed zone below 4 deg";
  gc_DbmTranslation_de_Text831 : WSTRING(36) := "Turret in Low Speed zone below 6 deg";
  gc_DbmTranslation_de_Text832 : WSTRING(57) := "Turret in Low Speed zone below 2 deg with basket rotation";
  gc_DbmTranslation_de_Text833 : WSTRING(57) := "Turret in Low Speed zone below 4 deg with basket rotation";
  gc_DbmTranslation_de_Text834 : WSTRING(57) := "Turret in Low Speed zone below 6 deg with basket rotation";
  gc_DbmTranslation_de_Text835 : WSTRING(43) := "Prevention for Limit Speed Acces Site Speed";
  gc_DbmTranslation_de_Text836 : WSTRING(37) := "Prevention for Limit Speed High Speed";
  gc_DbmTranslation_de_Text837 : WSTRING(36) := "Prevention for Limit Speed Low Speed";
  gc_DbmTranslation_de_Text838 : WSTRING(41) := "Prevention for Limit Low Speed Brake Test";
  gc_DbmTranslation_de_Text839 : WSTRING(35) := "Prevention exceeding of limit speed";
  gc_DbmTranslation_de_Text840 : WSTRING(54) := "Authorize global low speed in add performance function";
  gc_DbmTranslation_de_Text841 : WSTRING(51) := "N cycles brake need to make a validation brake test";
  gc_DbmTranslation_de_Text842 : WSTRING(40) := "N cycles critical , limit speed to 3km/h";
  gc_DbmTranslation_de_Text843 : WSTRING(44) := "Speed mini treshold to increment brake cycle";
  gc_DbmTranslation_de_Text844 : WSTRING(41) := "Pressure treshold for osci service brake ";
  gc_DbmTranslation_de_Text845 : WSTRING(41) := "Pressure treshold for fixe service brake ";
  gc_DbmTranslation_de_Text846 : WSTRING(40) := "Pressure treshold for osci parking brake";
  gc_DbmTranslation_de_Text847 : WSTRING(40) := "Pressure treshold for fixe parking brake";
  gc_DbmTranslation_de_Text848 : WSTRING(38) := "Time for osci service brake valid test";
  gc_DbmTranslation_de_Text849 : WSTRING(38) := "Time for fixe service brake valid test";
  gc_DbmTranslation_de_Text850 : WSTRING(38) := "Time for osci parking brake valid test";
  gc_DbmTranslation_de_Text851 : WSTRING(38) := "Time for fixe parking brake valid test";
  gc_DbmTranslation_de_Text852 : WSTRING(33) := "Speed mini to brake automatically";
  gc_DbmTranslation_de_Text853 : WSTRING(41) := "Valid condition to enable test brake time";
  gc_DbmTranslation_de_Text854 : WSTRING(45) := "Number element of delta transmission pressure";
  gc_DbmTranslation_de_Text855 : WSTRING(31) := "Seuil maximum de cycle de frein";
  gc_DbmTranslation_de_Text856 : WSTRING(33) := "2nd Seuil de dépassement critique";
  gc_DbmTranslation_de_Text857 : WSTRING(38) := "Temps pour la validation du test frein";
  gc_DbmTranslation_de_Text858 : WSTRING(38) := "Temps pour la validation du test frein";
  gc_DbmTranslation_de_Text859 : WSTRING(32) := "Threshold counter 2nd Park Brake";
  gc_DbmTranslation_de_Text860 : WSTRING(39) := "Minimum Threshold Active 2nd Park Brake";
  gc_DbmTranslation_de_Text861 : WSTRING(48) := "Fordid camera display when brake test is running";
  gc_DbmTranslation_de_Text862 : WSTRING(24) := "Pressure efficiency rate";
  gc_DbmTranslation_de_Text863 : WSTRING(34) := "Wich brake test selected on screen";
  gc_DbmTranslation_de_Text864 : WSTRING(68) := "Flag when cycle brake perform is over parameters NCycleNeedBrakeTest";
  gc_DbmTranslation_de_Text865 : WSTRING(67) := "Flag when cycle brake perform is over critial number of cycle brake";
  gc_DbmTranslation_de_Text866 : WSTRING(19) := "Up position of axle";
  gc_DbmTranslation_de_Text867 : WSTRING(21) := "Down position of axle";
  gc_DbmTranslation_de_Text868 : WSTRING(58) := "Incoherence position axle and test mode in rail or offrail";
  gc_DbmTranslation_de_Text869 : WSTRING(34) := "Test brake in rail or offrail mode";
  gc_DbmTranslation_de_Text870 : WSTRING(28) := "Flag when brake test running";
  gc_DbmTranslation_de_Text871 : WSTRING(34) := "Flag when valid brake test is done";
  gc_DbmTranslation_de_Text872 : WSTRING(49) := "enable condition to increment cycke brake perform";
  gc_DbmTranslation_de_Text873 : WSTRING(67) := "flag when a valid test brake is operared on oscillant service brake";
  gc_DbmTranslation_de_Text874 : WSTRING(62) := "flag when a valid test brake is operared on fixe service brake";
  gc_DbmTranslation_de_Text875 : WSTRING(67) := "flag when a valid test brake is operared on oscillant parking brake";
  gc_DbmTranslation_de_Text876 : WSTRING(62) := "flag when a valid test brake is operared on fixe parking brake";
  gc_DbmTranslation_de_Text877 : WSTRING(47) := "Simulation osci service breake select on screen";
  gc_DbmTranslation_de_Text878 : WSTRING(47) := "Simulation fixe service breake select on screen";
  gc_DbmTranslation_de_Text879 : WSTRING(47) := "Simulation osci parking breake select on screen";
  gc_DbmTranslation_de_Text880 : WSTRING(47) := "Simulation fixe parking breake select on screen";
  gc_DbmTranslation_de_Text881 : WSTRING(46) := "Simulation two service breake select on screen";
  gc_DbmTranslation_de_Text882 : WSTRING(46) := "Simulation two parking breake select on screen";
  gc_DbmTranslation_de_Text883 : WSTRING(39) := "Retain postition of joystick advanement";
  gc_DbmTranslation_de_Text884 : WSTRING(38) := "Actual postion of joystick advancement";
  gc_DbmTranslation_de_Text885 : WSTRING(29) := "Force oscillant service brake";
  gc_DbmTranslation_de_Text886 : WSTRING(24) := "Force fixe service brake";
  gc_DbmTranslation_de_Text887 : WSTRING(29) := "Force oscillant parking brake";
  gc_DbmTranslation_de_Text888 : WSTRING(24) := "Force fixe parking brake";
  gc_DbmTranslation_de_Text889 : WSTRING(35) := "stop all movement when a brake test";
  gc_DbmTranslation_de_Text890 : WSTRING(94) := "Authorize translation rail when nacelle in transport mode and no incohrence with axle position";
  gc_DbmTranslation_de_Text891 : WSTRING(38) := "Delta of transmission 1 and 2 preussre";
  gc_DbmTranslation_de_Text892 : WSTRING(38) := "Valid condition enable test brake flag";
  gc_DbmTranslation_de_Text893 : WSTRING(58) := "Flag when time out of valid condition to enable test brake";
  gc_DbmTranslation_de_Text894 : WSTRING(20) := "Pourcent cycle brake";
  gc_DbmTranslation_de_Text895 : WSTRING(18) := "Activation de l’EV";
  gc_DbmTranslation_de_Text896 : WSTRING(18) := "Activation de l’EV";
  gc_DbmTranslation_de_Text897 : WSTRING(76) := "Validation du test frein du frein de parc additionnel sur l’essieu Oscillant";
  gc_DbmTranslation_de_Text898 : WSTRING(71) := "Validation du test frein du frein de parc additionnel sur l’essieu Fixe";
  gc_DbmTranslation_de_Text899 : WSTRING(62) := "Variable de conversion du nombres de test frein en pourcentage";
  gc_DbmTranslation_de_Text900 : WSTRING(46) := "Variable de dépassement du seuil de test frein";
  gc_DbmTranslation_de_Text901 : WSTRING(55) := "Variable de dépassement du seuil critique de test frein";
  gc_DbmTranslation_de_Text902 : WSTRING(29) := "Additionnal Park Brake Active";
  gc_DbmTranslation_de_Text903 : WSTRING(30) := "Park Brake 2nd Pressure Active";
  gc_DbmTranslation_de_Text904 : WSTRING(66) := "Minimum allowed turret angle for the consistency check in ALO mode";
  gc_DbmTranslation_de_Text905 : WSTRING(66) := "Maximum allowed turret angle for the consistency check in ALO mode";
  gc_DbmTranslation_de_Text906 : WSTRING(72) := "Minimum allowed turret angle for the consistency check in multilane mode";
  gc_DbmTranslation_de_Text907 : WSTRING(72) := "Maximum allowed turret angle for the consistency check in multilane mode";
  gc_DbmTranslation_de_Text908 : WSTRING(55) := "ALO mode - Rear zone threshold of the turret (absolute)";
  gc_DbmTranslation_de_Text909 : WSTRING(81) := "ALO mode - Hysteresis applied on the rear zone threshold of the turret (relative)";
  gc_DbmTranslation_de_Text910 : WSTRING(114) := "ALO mode - Threshold use to reduce speed before the rear zone of the turret (relative to the front zone threshold)";
  gc_DbmTranslation_de_Text911 : WSTRING(56) := "ALO mode - Front zone threshold of the turret (absolute)";
  gc_DbmTranslation_de_Text912 : WSTRING(82) := "ALO mode - Hysteresis applied on the front zone threshold of the turret (relative)";
  gc_DbmTranslation_de_Text913 : WSTRING(115) := "ALO mode - Threshold use to reduce speed before the front zone of the turret (relative to the front zone threshold)";
  gc_DbmTranslation_de_Text914 : WSTRING(66) := "ALO mode - Threshold of the lower zone of the arrow arm (absolute)";
  gc_DbmTranslation_de_Text915 : WSTRING(85) := "ALO mode - Hysteresis applied on the lower zone threshold of the arrow arm (relative)";
  gc_DbmTranslation_de_Text916 : WSTRING(118) := "ALO mode - Threshold use to reduce speed before the lower zone of the arrow arm (relative to the lower zone threshold)";
  gc_DbmTranslation_de_Text917 : WSTRING(52) := "ALO mode - Turret rear end stop threshold (absolute)";
  gc_DbmTranslation_de_Text918 : WSTRING(78) := "ALO mode - Hysteresis applied on the turret rear end stop threshold (relative)";
  gc_DbmTranslation_de_Text919 : WSTRING(121) := "ALO mode - Threshold use to reduce speed before the rear end stop of the turret (relative to the rear end stop threshold)";
  gc_DbmTranslation_de_Text920 : WSTRING(52) := "ALO mode - Turret rear end stop threshold (absolute)";
  gc_DbmTranslation_de_Text921 : WSTRING(78) := "ALO mode - Hysteresis applied on the turret rear end stop threshold (relative)";
  gc_DbmTranslation_de_Text922 : WSTRING(121) := "ALO mode - Threshold use to reduce speed before the rear end stop of the turret (relative to the rear end stop threshold)";
  gc_DbmTranslation_de_Text923 : WSTRING(111) := "ALO mode - Threshold use to stop the turret before reaching the rear zone (relative to the rear zone threshold)";
  gc_DbmTranslation_de_Text924 : WSTRING(86) := "ALO mode - Hysteresis applied to the rear zone stop threshold of the turret (relative)";
  gc_DbmTranslation_de_Text925 : WSTRING(113) := "ALO mode - Threshold use to stop the turret before reaching the front zone (relative to the front zone threshold)";
  gc_DbmTranslation_de_Text926 : WSTRING(87) := "ALO mode - Hysteresis applied to the front zone stop threshold of the turret (relative)";
  gc_DbmTranslation_de_Text927 : WSTRING(116) := "ALO mode - Threshold use to stop the arrow arm before reaching the lower zone (relative to the lower zone threshold)";
  gc_DbmTranslation_de_Text928 : WSTRING(90) := "ALO mode - Hysteresis applied to the lower zone stop threshold of the arrow arm (relative)";
  gc_DbmTranslation_de_Text929 : WSTRING(34) := "Rail work mode selected by the key";
  gc_DbmTranslation_de_Text930 : WSTRING(59) := "Consistency check - wrong turret abutment in bilateral mode";
  gc_DbmTranslation_de_Text931 : WSTRING(59) := "Consistency check - wrong turret abutment in multilane mode";
  gc_DbmTranslation_de_Text932 : WSTRING(53) := "Consistency check - wrong turret abutment in ALO mode";
  gc_DbmTranslation_de_Text933 : WSTRING(77) := "Consistency check - wrong basket abutment in bilateral mode (only for France)";
  gc_DbmTranslation_de_Text934 : WSTRING(77) := "Consistency check - wrong basket abutment in multilane mode (only for France)";
  gc_DbmTranslation_de_Text935 : WSTRING(71) := "Consistency check - wrong basket abutment in ALO mode (only for France)";
  gc_DbmTranslation_de_Text936 : WSTRING(43) := "Consistency check - wrong abutment detected";
  gc_DbmTranslation_de_Text937 : WSTRING(59) := "Consistency check - wrong turret position in multilane mode";
  gc_DbmTranslation_de_Text938 : WSTRING(59) := "Consistency check - wrong basket position in multilane mode";
  gc_DbmTranslation_de_Text939 : WSTRING(53) := "Consistency check - wrong turret position in ALO mode";
  gc_DbmTranslation_de_Text940 : WSTRING(43) := "Consistency check - wrong position detected";
  gc_DbmTranslation_de_Text941 : WSTRING(49) := "Reduce the speed of the turret clockwise movement";
  gc_DbmTranslation_de_Text942 : WSTRING(57) := "Reduce the speed of the turret counter clockwise movement";
  gc_DbmTranslation_de_Text943 : WSTRING(47) := "Reduce the speed of the arrow arm down movement";
  gc_DbmTranslation_de_Text944 : WSTRING(34) := "Stop the turret clockwise movement";
  gc_DbmTranslation_de_Text945 : WSTRING(42) := "Stop the turret counter clockwise movement";
  gc_DbmTranslation_de_Text946 : WSTRING(34) := "Stop the basket clockwise movement";
  gc_DbmTranslation_de_Text947 : WSTRING(42) := "Stop the basket counter clockwise movement";
  gc_DbmTranslation_de_Text948 : WSTRING(32) := "Stop the arrow arm down movement";
  gc_DbmTranslation_de_Text949 : WSTRING(31) := "Stop the telescope out movement";
  gc_DbmTranslation_de_Text950 : WSTRING(23) := "Turret in the rear zone";
  gc_DbmTranslation_de_Text951 : WSTRING(24) := "Turret in the front zone";
  gc_DbmTranslation_de_Text952 : WSTRING(27) := "Arrow arm in the lower zone";
  gc_DbmTranslation_de_Text953 : WSTRING(60) := "Test variable for simulation - french version of the vehicle";
  gc_DbmTranslation_de_Text954 : WSTRING(57) := "Test variable for simulation - basket abutment track side";
  gc_DbmTranslation_de_Text955 : WSTRING(60) := "Test variable for simulation - basket abutment centered side";
  gc_DbmTranslation_de_Text956 : WSTRING(54) := "Test variable for simulation - basket left side sensor";
  gc_DbmTranslation_de_Text957 : WSTRING(55) := "Test variable for simulation - basket right side sensor";
  gc_DbmTranslation_de_Text958 : WSTRING(49) := "Test variable for simulation - telescop in sensor";
  gc_DbmTranslation_de_Text959 : WSTRING(54) := "Test variable for simulation - turret angular position";
  gc_DbmTranslation_de_Text960 : WSTRING(57) := "Test variable for simulation - arrow arm angular position";
  gc_DbmTranslation_de_Text961 : WSTRING(42) := "Abutment work mode selected by the sensors";
  gc_DbmTranslation_de_Text962 : WSTRING(0) := "";
  gc_DbmTranslation_de_Text963 : WSTRING(0) := "";
  gc_DbmTranslation_de_Text964 : WSTRING(0) := "";
  gc_DbmTranslation_de_Text965 : WSTRING(52) := "Delta arm treshold position for chenillard transport";
  gc_DbmTranslation_de_Text966 : WSTRING(54) := "Delta arm hysteresis position for chenillard transport";
  gc_DbmTranslation_de_Text967 : WSTRING(50) := "Arrow arm treshold position for off rail transport";
  gc_DbmTranslation_de_Text968 : WSTRING(52) := "Arrow arm hysteresis position for off rail transport";
  gc_DbmTranslation_de_Text969 : WSTRING(21) := "Turret angle thresold";
  gc_DbmTranslation_de_Text970 : WSTRING(64) := "Bouton on screen to seleted the off rail mode for break in brake";
  gc_DbmTranslation_de_Text971 : WSTRING(29) := "Force oscillant service brake";
  gc_DbmTranslation_de_Text972 : WSTRING(24) := "Force fixe service brake";
  gc_DbmTranslation_de_Text973 : WSTRING(29) := "Force oscillant parking brake";
  gc_DbmTranslation_de_Text974 : WSTRING(24) := "Force fixe parking brake";
  gc_DbmTranslation_de_Text975 : WSTRING(49) := "Stop all movement when a break in brake is during";
  gc_DbmTranslation_de_Text976 : WSTRING(58) := "Incoherence position axle and test mode in rail or offrail";
  gc_DbmTranslation_de_Text977 : WSTRING(53) := "Advancement period, reset every new advancement order";
  gc_DbmTranslation_de_Text978 : WSTRING(22) := "Break in brake running";
  gc_DbmTranslation_de_Text979 : WSTRING(47) := "Simu oscillant service brake selected on screen";
  gc_DbmTranslation_de_Text980 : WSTRING(42) := "Simu fixe service brake selected on screen";
  gc_DbmTranslation_de_Text981 : WSTRING(40) := "Simu 2 service brakes selected on screen";
  gc_DbmTranslation_de_Text982 : WSTRING(47) := "Authorize transaltion on rail by break in brake";
  gc_DbmTranslation_de_Text983 : WSTRING(32) := "Service brake selected on screen";
  gc_DbmTranslation_de_Text984 : WSTRING(26) := "Advacnement period by 10ms";
  gc_DbmTranslation_de_Text985 : WSTRING(30) := "Osci service brake in brake On";
  gc_DbmTranslation_de_Text986 : WSTRING(30) := "Fixe service brake in brake On";
  gc_DbmTranslation_de_Text987 : WSTRING(30) := "Both service brake in brake On";
  gc_DbmTranslation_de_Text988 : WSTRING(36) := "Post selected to control the vehicle";
  gc_DbmTranslation_de_Text989 : WSTRING(17) := "Enable the buzzer";
  gc_DbmTranslation_de_Text990 : WSTRING(16) := "The slope is low";
  gc_DbmTranslation_de_Text991 : WSTRING(17) := "The slope is high";
  gc_DbmTranslation_de_Text992 : WSTRING(45) := "All commands of the nacelle post are disabled";
  gc_DbmTranslation_de_Text993 : WSTRING(51) := "All commands of the radio command post are disabled";
  gc_DbmTranslation_de_Text994 : WSTRING(44) := "All commands of the turret post are disabled";
  gc_DbmTranslation_de_Text995 : WSTRING(41) := "Variable used to simulate the slope angle";
  gc_DbmTranslation_de_Text996 : WSTRING(50) := "All ouput consigne of transaltion rail is disabled";
  gc_DbmTranslation_de_Text997 : WSTRING(32) := "Authorise radio element position";
  gc_DbmTranslation_de_Text998 : WSTRING(43) := "Threshold use to detect if the slope is low";
  gc_DbmTranslation_de_Text999 : WSTRING(56) := "Hysteresis applied on the slope low threshold (relative)";
  gc_DbmTranslation_de_Text1000 : WSTRING(44) := "Threshold use to detect if the slope is high";
  gc_DbmTranslation_de_Text1001 : WSTRING(57) := "Hysteresis applied on the slope high threshold (relative)";
  gc_DbmTranslation_de_Text1002 : WSTRING(26) := "Slope crawler max treshold";
  gc_DbmTranslation_de_Text1003 : WSTRING(33) := "Life byte sent to the controllers";
  gc_DbmTranslation_de_Text1004 : WSTRING(35) := "Delta arm move up button is pressed";
  gc_DbmTranslation_de_Text1005 : WSTRING(37) := "Delta arm move down button is pressed";
  gc_DbmTranslation_de_Text1006 : WSTRING(35) := "Arrow arm move up button is pressed";
  gc_DbmTranslation_de_Text1007 : WSTRING(37) := "Arrow arm move down button is pressed";
  gc_DbmTranslation_de_Text1008 : WSTRING(34) := "Pendular move up button is pressed";
  gc_DbmTranslation_de_Text1009 : WSTRING(36) := "Pendular move down button is pressed";
  gc_DbmTranslation_de_Text1010 : WSTRING(36) := "Telescope move out button is pressed";
  gc_DbmTranslation_de_Text1011 : WSTRING(35) := "Telescope move in button is pressed";
  gc_DbmTranslation_de_Text1012 : WSTRING(44) := "Basket inclinaison move up button is pressed";
  gc_DbmTranslation_de_Text1013 : WSTRING(46) := "Basket inclinaison move down button is pressed";
  gc_DbmTranslation_de_Text1014 : WSTRING(41) := "Rotate turret clockwise button is pressed";
  gc_DbmTranslation_de_Text1015 : WSTRING(49) := "Rotate turret counter clockwise button is pressed";
  gc_DbmTranslation_de_Text1016 : WSTRING(41) := "Basket rotation move up button is pressed";
  gc_DbmTranslation_de_Text1017 : WSTRING(43) := "Basket rotation move down button is pressed";
  gc_DbmTranslation_de_Text1018 : WSTRING(23) := "Key RPM Selection level";
  gc_DbmTranslation_de_Text1019 : WSTRING(32) := "Key Desactivation RPM selection ";
  gc_DbmTranslation_de_Text1020 : WSTRING(51) := "Activation forcing White Rail lights Front and Rear";
  gc_DbmTranslation_de_Text1021 : WSTRING(16) := "Activation neons";
  gc_DbmTranslation_de_Text1022 : WSTRING(19) := "Key Calibration Min";
  gc_DbmTranslation_de_Text1023 : WSTRING(19) := "Key Calibration Max";
  gc_DbmTranslation_de_Text1024 : WSTRING(26) := "Key Calibration Validation";
  gc_DbmTranslation_de_Text1025 : WSTRING(89) := "Element choice 1=Telescope; 2=Arrow arm; 3=Delta arm; 4=Turret; 5=Slope; 6=Measuring Mast";
  gc_DbmTranslation_de_Text1026 : WSTRING(27) := "Key Calibration Max (-180°)";
  gc_DbmTranslation_de_Text1027 : WSTRING(28) := "Key Slope Longitudinal reset";
  gc_DbmTranslation_de_Text1028 : WSTRING(27) := "Key Slope Transversal reset";
  gc_DbmTranslation_de_Text1029 : WSTRING(76) := "DM_HIGH_HYDRAULIC_TEMP_CRAWLER - Overflow Threshold Fault Temperature Tracks";
  gc_DbmTranslation_de_Text1030 : WSTRING(71) := "DM_HIGH_HYDRAULIC_TEMP_RAIL - Overflow Threshold Fault Temperature Rail";
  gc_DbmTranslation_de_Text1031 : WSTRING(77) := "DM_ALARM_HYDRAULIC_TEMP_CRAWLER - Overflow Threshold Alarm Temperature Tracks";
  gc_DbmTranslation_de_Text1032 : WSTRING(72) := "DM_ALARM_HYDRAULIC_TEMP_RAIL - Overflow Threshold Alarm Temperature Rail";
  gc_DbmTranslation_de_Text1033 : WSTRING(69) := "DM_ONE_SPEED_SENSOR_FAULT - Tolerenace Threshold both 2 speed sensors";
  gc_DbmTranslation_de_Text1034 : WSTRING(54) := "DM_SLOPE_FAULT - tolerance both 2 chanelles slope long";
  gc_DbmTranslation_de_Text1035 : WSTRING(71) := "DM_OSCILLANT_CIRCUIT_FAULT - block isccilation axle pressure Threshold ";
  gc_DbmTranslation_de_Text1036 : WSTRING(73) := "DM_OSCILLANT_CIRCUIT_FAULT - unblock isccilation axle pressure Threshold ";
  gc_DbmTranslation_de_Text1037 : WSTRING(76) := "DM_SERVICE_BRAKE_PRESSURE_FAULT - Min service brake pressure fault threshold";
  gc_DbmTranslation_de_Text1038 : WSTRING(76) := "DM_SERVICE_BRAKE_PRESSURE_FAULT - Max service brake pressure fault threshold";
  gc_DbmTranslation_de_Text1039 : WSTRING(55) := "DM_SLOPE_FAULT  - tolerance both 2 chanelles slope long";
  gc_DbmTranslation_de_Text1040 : WSTRING(79) := "DM_TRANS_CRAWLER_PRESSURE_HOOK - minimal pressure transmission when hook is off";
  gc_DbmTranslation_de_Text1041 : WSTRING(80) := "DM_TURRET_SENSOR_FAULT  - tolerence trehsold betwen 2 channels of turrent sensor";
  gc_DbmTranslation_de_Text1042 : WSTRING(108) := "DM_C0_OUT_OF_RANGE_JOY_DELTA_ARM_48XS - min alarm value of joytick delta arm in % according batterie voltage";
  gc_DbmTranslation_de_Text1043 : WSTRING(108) := "DM_C0_OUT_OF_RANGE_JOY_DELTA_ARM_48XS - max alarm value of joytick delta arm in % according batterie voltage";
  gc_DbmTranslation_de_Text1044 : WSTRING(108) := "DM_C0_OUT_OF_RANGE_JOY_ARROW_ARM_48XS - min alarm value of joytick arrow arm in % according batterie voltage";
  gc_DbmTranslation_de_Text1045 : WSTRING(108) := "DM_C0_OUT_OF_RANGE_JOY_ARROW_ARM_48XS - max alarm value of joytick arrow arm in % according batterie voltage";
  gc_DbmTranslation_de_Text1046 : WSTRING(116) := "DM_C0_OUT_OF_RANGE_JOY_TELESCOPE_ARM_48XS - min alarm value of joytick telescope arm in % according batterie voltage";
  gc_DbmTranslation_de_Text1047 : WSTRING(116) := "DM_C0_OUT_OF_RANGE_JOY_TELESCOPE_ARM_48XS - max alarm value of joytick telescope arm in % according batterie voltage";
  gc_DbmTranslation_de_Text1048 : WSTRING(123) := "DM_C0_OUT_OF_RANGE_JOY_ROT_TURRET_ARM_48XS - min alarm value of joytick rotation turret arm in % according batterie voltage";
  gc_DbmTranslation_de_Text1049 : WSTRING(123) := "DM_C0_OUT_OF_RANGE_JOY_ROT_TURRET_ARM_48XS - max alarm value of joytick rotation turret arm in % according batterie voltage";
  gc_DbmTranslation_de_Text1050 : WSTRING(120) := "DM_C0_OUT_OF_RANGE_JOY_ADVANCEMENT_48XS - min alarm value of joytick rotation turret arm in % according batterie voltage";
  gc_DbmTranslation_de_Text1051 : WSTRING(120) := "DM_C0_OUT_OF_RANGE_JOY_ADVANCEMENT_48XS - max alarm value of joytick rotation turret arm in % according batterie voltage";
  gc_DbmTranslation_de_Text1052 : WSTRING(61) := "DM_HIGH_HYDRAULIC_TEMP_RAIL - hysteresis treshold temperature";
  gc_DbmTranslation_de_Text1053 : WSTRING(43) := "Reduce track speed when temperature default";
  gc_DbmTranslation_de_Text1054 : WSTRING(82) := "Paramètre à ne jamais mettre à zéro. Utilisation pour le set du défaut de pression";
  gc_DbmTranslation_de_Text1055 : WSTRING(32) := "Activation de l’alarme de bypass";
  gc_DbmTranslation_de_Text1056 : WSTRING(17) := "Time Bypass Fault";
  gc_DbmTranslation_de_Text1057 : WSTRING(48) := "Threshold of thermic transmission pressure Alarm";
  gc_DbmTranslation_de_Text1058 : WSTRING(49) := "Threshold of electric transmission pressure Alarm";
  gc_DbmTranslation_de_Text1059 : WSTRING(60) := "Time detect for the alarm of the Thermic pump on Translation";
  gc_DbmTranslation_de_Text1060 : WSTRING(46) := "Time detect for the alarm of the Electric pump";
  gc_DbmTranslation_de_Text1061 : WSTRING(0) := "";
  gc_DbmTranslation_de_Text1062 : WSTRING(34) := "Fault on thermic pump transmission";
  gc_DbmTranslation_de_Text1063 : WSTRING(55) := "Time to detect the fault on the thermic pump are passed";
  gc_DbmTranslation_de_Text1064 : WSTRING(52) := "Active memorisation of the fault on the thermic pump";
  gc_DbmTranslation_de_Text1065 : WSTRING(22) := "Fault on electric pump";
  gc_DbmTranslation_de_Text1066 : WSTRING(56) := "Time to detect the fault on the electric pump are passed";
  gc_DbmTranslation_de_Text1067 : WSTRING(57) := "Active memorisation of the fault on the DMC electric pump";
  gc_DbmTranslation_de_Text1068 : WSTRING(40) := "Active fault on thermic or electric pump";
  gc_DbmTranslation_de_Text1069 : WSTRING(0) := "";
  gc_DbmTranslation_de_Text1070 : WSTRING(0) := "";
  gc_DbmTranslation_de_Text1071 : WSTRING(0) := "";
  gc_DbmTranslation_de_Text1072 : WSTRING(0) := "";
  gc_DbmTranslation_de_Text1073 : WSTRING(0) := "";
  gc_DbmTranslation_de_Text1074 : WSTRING(50) := "Last error code returned by the UART Init function";
  gc_DbmTranslation_de_Text1075 : WSTRING(51) := "Last error code returned by the UART Write function";
  gc_DbmTranslation_de_Text1076 : WSTRING(68) := "Successfully queued data butes (returned by the UART Write fucntion)";
  gc_DbmTranslation_de_Text1077 : WSTRING(17) := "Displayed digit 1";
  gc_DbmTranslation_de_Text1078 : WSTRING(17) := "Displayed digit 2";
  gc_DbmTranslation_de_Text1079 : WSTRING(17) := "Displayed digit 3";
  gc_DbmTranslation_de_Text1080 : WSTRING(17) := "Displayed digit 4";
  gc_DbmTranslation_de_Text1081 : WSTRING(43) := "Data array given to the UART Write function";
  gc_DbmTranslation_de_Text1082 : WSTRING(43) := "Data array given to the UART Write function";
  gc_DbmTranslation_de_Text1083 : WSTRING(43) := "Data array given to the UART Write function";
  gc_DbmTranslation_de_Text1084 : WSTRING(43) := "Data array given to the UART Write function";
  gc_DbmTranslation_de_Text1085 : WSTRING(43) := "Data array given to the UART Write function";
  gc_DbmTranslation_de_Text1086 : WSTRING(43) := "Data array given to the UART Write function";
  gc_DbmTranslation_de_Text1087 : WSTRING(43) := "Data array given to the UART Write function";
  gc_DbmTranslation_de_Text1088 : WSTRING(43) := "Data array given to the UART Write function";
  gc_DbmTranslation_de_Text1089 : WSTRING(43) := "Data array given to the UART Write function";
  gc_DbmTranslation_de_Text1090 : WSTRING(91) := "Refresh cycle time or the mast digital display ( cycle time of the message sent to display)";
  gc_DbmTranslation_de_Text1091 : WSTRING(0) := "";
  gc_DbmTranslation_de_Text1092 : WSTRING(0) := "";
  gc_DbmTranslation_de_Text1093 : WSTRING(0) := "";
  gc_DbmTranslation_de_Text1094 : WSTRING(0) := "";
  gc_DbmTranslation_de_Text1095 : WSTRING(0) := "";
  gc_DbmTranslation_de_Text1096 : WSTRING(0) := "";
  gc_DbmTranslation_de_Text1097 : WSTRING(0) := "";
